SPLINE
SPL {X  -159.990, Y  +497.800, Z    +0.000, E1   +31.845, E3 +413374.245}
SPL {X  -159.990, Y  +492.180, Z    +0.000, E1   +32.851, E3 +413386.381}
SPL {X  -159.990, Y  +486.073, Z    +0.000, E1   +33.960, E3 +413399.016}
SPL {X  -159.990, Y  +477.314, Z    +0.000, E1   +35.342, E3 +413417.195}
SPL {X  -159.990, Y  +471.459, Z    +0.000, E1   +35.779, E3 +413431.734}
SPL {X  -159.990, Y  +467.485, Z    +0.000, E1   +35.768, E3 +413443.464}
SPL {X  -159.990, Y  +462.739, Z    +0.000, E1   +35.799, E3 +413457.392}
SPL {X  -159.990, Y  +457.385, Z    +0.000, E1   +35.788, E3 +413473.175}
SPL {X  -159.990, Y  +452.637, Z    +0.000, E1   +35.783, E3 +413487.167}
SPL {X  -159.990, Y  +448.227, Z    +0.000, E1   +35.776, E3 +413500.163}
SPL {X  -159.990, Y  +443.707, Z    +0.000, E1   +35.784, E3 +413513.459}
SPL {X  -159.990, Y  +439.109, Z    +0.000, E1   +35.781, E3 +413526.995}
SPL {X  -159.990, Y  +434.400, Z    +0.000, E1   +35.789, E3 +413540.849}
SPL {X  -159.990, Y  +430.115, Z    +0.000, E1   +35.777, E3 +413553.466}
SPL {X  -159.990, Y  +425.407, Z    +0.000, E1   +35.800, E3 +413567.306}
SPL {X  -159.990, Y  +420.199, Z    +0.000, E1   +35.790, E3 +413582.660}
SPL {X  -159.990, Y  +414.514, Z    +0.000, E1   +35.815, E3 +413599.359}
SPL {X  -159.990, Y  +408.600, Z    +0.000, E1   +35.802, E3 +413616.798}
SPL {X  -159.990, Y  +403.496, Z    +0.000, E1   +35.787, E3 +413631.852}
SPL {X  -159.990, Y  +398.606, Z    +0.000, E1   +35.794, E3 +413646.240}
SPL {X  -159.990, Y  +394.138, Z    +0.000, E1   +35.778, E3 +413659.423}
SPL {X  -159.990, Y  +388.813, Z    +0.000, E1   +35.819, E3 +413675.035}
SPL {X  -159.990, Y  +383.172, Z    +0.000, E1   +35.789, E3 +413691.689}
SPL {X  -159.936, Y  +378.352, Z    +0.000, E1   +35.782, E3 +413705.928}
SPL {X  -159.693, Y  +372.749, Z    +0.000, E1   +35.767, E3 +413722.660}
SPL {X  -159.203, Y  +366.647, Z    +0.000, E1   +35.680, E3 +413741.146}
SPL {X  -158.715, Y  +362.338, Z    +0.000, E1   +35.547, E3 +413754.451}
SPL {X  -158.237, Y  +358.884, Z    +0.000, E1   +35.480, E3 +413765.108}
SPL {X  -157.724, Y  +355.670, Z    +0.000, E1   +35.371, E3 +413775.142}
SPL {X  -157.185, Y  +352.671, Z    +0.000, E1   +35.292, E3 +413784.521}
SPL {X  -156.302, Y  +348.345, Z    +0.000, E1   +35.165, E3 +413798.142}
SPL {X  -155.054, Y  +343.066, Z    +0.000, E1   +34.964, E3 +413814.956}
SPL {X  -154.305, Y  +340.232, Z    +0.000, E1   +28.975, E3 +413872.516}
ENDSPLINE

SPLINE
SPL {X  -158.456, Y  +360.399, Z    +0.000, E1   +16.490, E3 +413909.336}
SPL {X  -159.553, Y  +370.677, Z    +0.000, E1   +10.576, E3 +413917.096}
SPL {X  -159.960, Y  +379.402, Z    +0.000, E1    +5.303, E3 +413921.116}
SPL {X  -159.990, Y  +387.301, Z    +0.000, E1    +0.001, E3 +413923.578}
SPL {X  -159.990, Y  +392.161, Z    +0.000, E1    -3.946, E3 +413924.989}
SPL {X  -159.990, Y  +396.375, Z    +0.000, E1    -7.538, E3 +413926.411}
SPL {X  -159.990, Y  +404.277, Z    +0.000, E1   -14.543, E3 +413930.075}
SPL {X  -159.990, Y  +423.101, Z    +0.000, E1   -27.351, E3 +413946.513}
SPL {X  -159.990, Y  +430.933, Z    +0.000, E1   -30.672, E3 +413956.484}
SPL {X  -159.990, Y  +451.842, Z    +0.000, E1   -35.050, E3 +413995.856}
SPL {X  -159.990, Y  +456.402, Z    +0.000, E1   -35.061, E3 +414009.632}
SPL {X  -159.990, Y  +460.708, Z    +0.000, E1   -35.045, E3 +414022.689}
SPL {X  -159.990, Y  +464.162, Z    +0.000, E1   -35.038, E3 +414033.146}
SPL {X  -159.990, Y  +467.857, Z    +0.000, E1   -35.053, E3 +414044.303}
SPL {X  -159.990, Y  +471.326, Z    +0.000, E1   -35.038, E3 +414054.798}
SPL {X  -159.990, Y  +474.610, Z    +0.000, E1   -35.053, E3 +414064.697}
SPL {X  -159.990, Y  +478.303, Z    +0.000, E1   -35.049, E3 +414075.869}
SPL {X  -159.990, Y  +482.537, Z    +0.000, E1   -35.066, E3 +414088.661}
SPL {X  -159.990, Y  +487.181, Z    +0.000, E1   -35.054, E3 +414102.744}
SPL {X  -159.990, Y  +492.368, Z    +0.000, E1   -35.076, E3 +414118.415}
SPL {X  -159.990, Y  +497.072, Z    +0.000, E1   -35.040, E3 +414132.712}
SPL {X  -159.990, Y  +501.645, Z    +0.000, E1   -35.067, E3 +414146.495}
SPL {X  -159.990, Y  +506.307, Z    +0.000, E1   -35.049, E3 +414160.617}
SPL {X  -159.990, Y  +511.643, Z    +0.000, E1   -35.091, E3 +414176.697}
SPL {X  -159.990, Y  +517.156, Z    +0.000, E1   -35.059, E3 +414193.415}
SPL {X  -159.990, Y  +521.637, Z    +0.000, E1   -35.056, E3 +414206.978}
SPL {X  -159.990, Y  +526.246, Z    +0.000, E1   -35.065, E3 +414220.882}
SPL {X  -159.990, Y  +530.289, Z    +0.000, E1   -35.044, E3 +414233.168}
SPL {X  -159.990, Y  +534.797, Z    +0.000, E1   -35.069, E3 +414246.768}
SPL {X  -159.990, Y  +538.710, Z    +0.000, E1   -35.033, E3 +414258.665}
SPL {X  -159.990, Y  +542.114, Z    +0.000, E1   -35.053, E3 +414268.917}
SPL {X  -159.990, Y  +545.724, Z    +0.000, E1   -35.043, E3 +414279.842}
SPL {X  -159.990, Y  +549.546, Z    +0.000, E1   -35.061, E3 +414291.366}
SPL {X  -159.990, Y  +554.793, Z    +0.000, E1   -35.100, E3 +414307.129}
SPL {X  -159.990, Y  +560.931, Z    +0.000, E1   -35.098, E3 +414325.691}
SPL {X  -159.990, Y  +566.542, Z    +0.000, E1   -35.080, E3 +414342.699}
SPL {X  -159.990, Y  +570.261, Z    +0.000, E1   -35.046, E3 +414353.995}
SPL {X  -159.990, Y  +574.780, Z    +0.000, E1   -35.101, E3 +414367.574}
SPL {X  -159.990, Y  +580.750, Z    +0.000, E1   -35.087, E3 +414385.650}
SPL {X  -159.990, Y  +585.414, Z    +0.000, E1   -35.059, E3 +414399.796}
SPL {X  -159.990, Y  +588.716, Z    +0.000, E1   -35.047, E3 +414409.799}
SPL {X  -159.990, Y  +592.923, Z    +0.000, E1   -35.084, E3 +414422.463}
SPL {X  -159.990, Y  +598.554, Z    +0.000, E1   -35.088, E3 +414439.483}
SPL {X  -159.990, Y  +603.289, Z    +0.000, E1   -35.068, E3 +414453.810}
SPL {X  -159.990, Y  +606.793, Z    +0.000, E1   -35.050, E3 +414464.452}
SPL {X  -159.990, Y  +611.113, Z    +0.000, E1   -35.087, E3 +414477.443}
SPL {X  -159.990, Y  +616.690, Z    +0.000, E1   -35.089, E3 +414494.306}
SPL {X  -159.990, Y  +621.534, Z    +0.000, E1   -35.068, E3 +414508.965}
SPL {X  -159.990, Y  +625.237, Z    +0.000, E1   -35.062, E3 +414520.167}
SPL {X  -159.990, Y  +629.217, Z    +0.000, E1   -35.065, E3 +414532.225}
SPL {X  -159.990, Y  +632.566, Z    +0.000, E1   -35.044, E3 +414542.387}
SPL {X  -159.990, Y  +636.917, Z    +0.000, E1   -35.095, E3 +414555.462}
SPL {X  -159.990, Y  +641.534, Z    +0.000, E1   -35.053, E3 +414569.489}
SPL {X  -159.990, Y  +645.423, Z    +0.000, E1   -35.070, E3 +414581.225}
SPL {X  -159.990, Y  +650.555, Z    +0.000, E1   -35.089, E3 +414596.714}
SPL {X  -159.990, Y  +656.270, Z    +0.000, E1   -35.087, E3 +414614.007}
SPL {X  -159.990, Y  +661.105, Z    +0.000, E1   -35.059, E3 +414628.671}
SPL {X  -159.990, Y  +665.311, Z    +0.000, E1   -35.064, E3 +414641.385}
SPL {X  -159.990, Y  +670.193, Z    +0.000, E1   -35.076, E3 +414656.133}
SPL {X  -159.948, Y  +675.148, Z    +0.000, E1   -35.069, E3 +414671.125}
SPL {X  -159.805, Y  +679.202, Z    +0.000, E1   -35.029, E3 +414683.557}
SPL {X  -159.584, Y  +682.885, Z    +0.000, E1   -34.997, E3 +414694.917}
SPL {X  -159.292, Y  +686.426, Z    +0.000, E1   -34.947, E3 +414705.919}
SPL {X  -158.886, Y  +690.264, Z    +0.000, E1   -34.888, E3 +414717.935}
SPL {X  -158.362, Y  +694.266, Z    +0.000, E1   -34.794, E3 +414730.609}
SPL {X  -157.614, Y  +698.973, Z    +0.000, E1   -34.690, E3 +414745.609}
SPL {X  -156.640, Y  +704.066, Z    +0.000, E1   -34.516, E3 +414762.034}
SPL {X  -155.835, Y  +707.723, Z    +0.000, E1   -34.344, E3 +414773.977}
SPL {X  -155.153, Y  +710.542, Z    +0.000, E1   -34.234, E3 +414783.196}
SPL {X  -153.767, Y  +715.686, Z    +0.000, E1   -30.747, E3 +414828.414}
ENDSPLINE

SPLINE
SPL {X  -155.537, Y  +708.983, Z    +0.000, E1   -25.008, E3 +414859.219}
SPL {X  -158.838, Y  +690.666, Z    +0.000, E1   -14.584, E3 +414883.932}
SPL {X  -159.750, Y  +680.262, Z    +0.000, E1    -8.563, E3 +414890.072}
SPL {X  -159.973, Y  +673.798, Z    +0.000, E1    -4.600, E3 +414892.536}
SPL {X  -159.990, Y  +667.448, Z    +0.000, E1    -0.356, E3 +414894.316}
SPL {X  -159.990, Y  +662.686, Z    +0.000, E1    +3.472, E3 +414895.551}
SPL {X  -159.990, Y  +657.071, Z    +0.000, E1    +8.297, E3 +414897.429}
SPL {X  -159.990, Y  +646.193, Z    +0.000, E1   +17.980, E3 +414903.156}
SPL {X  -159.990, Y  +621.124, Z    +0.000, E1   +32.598, E3 +414926.643}
SPL {X  -159.990, Y  +597.855, Z    +0.000, E1   +36.862, E3 +414969.562}
SPL {X  -159.990, Y  +592.884, Z    +0.000, E1   +36.865, E3 +414983.633}
SPL {X  -159.990, Y  +587.104, Z    +0.000, E1   +36.878, E3 +414999.990}
SPL {X  -159.990, Y  +581.795, Z    +0.000, E1   +36.847, E3 +415015.088}
SPL {X  -159.990, Y  +577.286, Z    +0.000, E1   +36.853, E3 +415027.845}
SPL {X  -159.990, Y  +572.409, Z    +0.000, E1   +36.854, E3 +415041.657}
SPL {X  -159.990, Y  +567.110, Z    +0.000, E1   +36.868, E3 +415056.619}
SPL {X  -159.990, Y  +562.387, Z    +0.000, E1   +36.853, E3 +415069.980}
SPL {X  -159.990, Y  +557.944, Z    +0.000, E1   +36.859, E3 +415082.574}
SPL {X  -159.990, Y  +553.661, Z    +0.000, E1   +36.844, E3 +415094.737}
SPL {X  -159.990, Y  +549.195, Z    +0.000, E1   +36.856, E3 +415107.373}
SPL {X  -159.990, Y  +544.733, Z    +0.000, E1   +36.845, E3 +415120.019}
SPL {X  -159.990, Y  +539.889, Z    +0.000, E1   +36.872, E3 +415133.703}
SPL {X  -159.990, Y  +534.469, Z    +0.000, E1   +36.855, E3 +415149.101}
SPL {X  -159.990, Y  +530.428, Z    +0.000, E1   +36.821, E3 +415160.634}
SPL {X  -159.990, Y  +527.151, Z    +0.000, E1   +36.828, E3 +415169.897}
SPL {X  -159.990, Y  +522.641, Z    +0.000, E1   +36.854, E3 +415182.629}
SPL {X  -159.990, Y  +517.225, Z    +0.000, E1   +36.859, E3 +415197.964}
SPL {X  -159.990, Y  +512.789, Z    +0.000, E1   +36.824, E3 +415210.591}
SPL {X  -159.990, Y  +508.591, Z    +0.000, E1   +36.846, E3 +415222.454}
SPL {X  -159.990, Y  +503.454, Z    +0.000, E1   +36.847, E3 +415237.009}
SPL {X  -159.990, Y  +498.507, Z    +0.000, E1   +36.487, E3 +415253.458}
ENDSPLINE

SPLINE
SPL {X  -159.990, Y  +506.994, Z    +0.000, E1   +30.162, E3 +415265.967}
ENDSPLINE

SPLINE
SPL {X  -159.990, Y  +502.084, Z    +0.000, E1   +31.057, E3 +415277.619}
SPL {X  -159.990, Y  +496.272, Z    +0.000, E1   +32.117, E3 +415290.610}
SPL {X  -159.990, Y  +492.180, Z    +0.000, E1   +32.851, E3 +415299.424}
SPL {X  -159.990, Y  +486.073, Z    +0.000, E1   +33.960, E3 +415312.060}
SPL {X  -159.990, Y  +477.314, Z    +0.000, E1   +35.342, E3 +415330.238}
SPL {X  -159.990, Y  +471.459, Z    +0.000, E1   +35.779, E3 +415344.778}
SPL {X  -159.990, Y  +467.485, Z    +0.000, E1   +35.768, E3 +415356.507}
SPL {X  -159.990, Y  +462.739, Z    +0.000, E1   +35.799, E3 +415370.435}
SPL {X  -159.990, Y  +457.385, Z    +0.000, E1   +35.788, E3 +415386.218}
SPL {X  -159.990, Y  +452.637, Z    +0.000, E1   +35.783, E3 +415400.210}
SPL {X  -159.990, Y  +448.227, Z    +0.000, E1   +35.776, E3 +415413.207}
SPL {X  -159.990, Y  +443.707, Z    +0.000, E1   +35.784, E3 +415426.502}
SPL {X  -159.990, Y  +439.109, Z    +0.000, E1   +35.781, E3 +415440.038}
SPL {X  -159.990, Y  +435.535, Z    +0.000, E1   +35.764, E3 +415450.589}
SPL {X  -159.990, Y  +431.100, Z    +0.000, E1   +35.807, E3 +415463.574}
SPL {X  -159.990, Y  +426.641, Z    +0.000, E1   +35.769, E3 +415476.760}
SPL {X  -159.990, Y  +422.627, Z    +0.000, E1   +35.788, E3 +415488.558}
SPL {X  -159.990, Y  +419.027, Z    +0.000, E1   +35.762, E3 +415499.198}
SPL {X  -159.990, Y  +414.514, Z    +0.000, E1   +35.815, E3 +415512.402}
SPL {X  -159.990, Y  +409.702, Z    +0.000, E1   +35.772, E3 +415526.643}
SPL {X  -159.990, Y  +404.413, Z    +0.000, E1   +35.821, E3 +415542.146}
SPL {X  -159.990, Y  +398.606, Z    +0.000, E1   +35.794, E3 +415559.283}
SPL {X  -159.990, Y  +394.138, Z    +0.000, E1   +35.778, E3 +415572.466}
SPL {X  -159.990, Y  +388.813, Z    +0.000, E1   +35.819, E3 +415588.078}
SPL {X  -159.990, Y  +383.172, Z    +0.000, E1   +35.789, E3 +415604.733}
SPL {X  -159.936, Y  +378.352, Z    +0.000, E1   +35.782, E3 +415618.972}
SPL {X  -159.790, Y  +374.497, Z    +0.000, E1   +35.735, E3 +415630.516}
SPL {X  -159.547, Y  +370.604, Z    +0.000, E1   +35.724, E3 +415642.201}
SPL {X  -159.134, Y  +365.969, Z    +0.000, E1   +35.644, E3 +415656.286}
SPL {X  -158.606, Y  +361.498, Z    +0.000, E1   +35.550, E3 +415670.051}
SPL {X  -157.918, Y  +356.833, Z    +0.000, E1   +35.439, E3 +415684.503}
SPL {X  -157.185, Y  +352.671, Z    +0.000, E1   +35.292, E3 +415697.564}
SPL {X  -156.302, Y  +348.345, Z    +0.000, E1   +35.165, E3 +415711.185}
SPL {X  -155.054, Y  +343.066, Z    +0.000, E1   +34.964, E3 +415728.000}
SPL {X  -154.305, Y  +340.232, Z    +0.000, E1   +28.975, E3 +415785.560}
ENDSPLINE

SPLINE
SPL {X  -158.456, Y  +360.399, Z    +0.000, E1   +16.490, E3 +415822.380}
SPL {X  -159.553, Y  +370.677, Z    +0.000, E1   +10.576, E3 +415830.140}
SPL {X  -159.960, Y  +379.402, Z    +0.000, E1    +5.303, E3 +415834.160}
SPL {X  -159.990, Y  +387.301, Z    +0.000, E1    +0.001, E3 +415836.621}
SPL {X  -159.990, Y  +392.161, Z    +0.000, E1    -3.946, E3 +415838.033}
SPL {X  -159.990, Y  +396.375, Z    +0.000, E1    -7.538, E3 +415839.455}
SPL {X  -159.990, Y  +404.277, Z    +0.000, E1   -14.543, E3 +415843.118}
SPL {X  -159.990, Y  +423.101, Z    +0.000, E1   -27.351, E3 +415859.557}
SPL {X  -159.990, Y  +430.933, Z    +0.000, E1   -30.672, E3 +415869.528}
SPL {X  -159.990, Y  +451.842, Z    +0.000, E1   -35.050, E3 +415908.899}
SPL {X  -159.990, Y  +456.402, Z    +0.000, E1   -35.061, E3 +415922.675}
SPL {X  -159.990, Y  +460.708, Z    +0.000, E1   -35.045, E3 +415935.733}
SPL {X  -159.990, Y  +464.162, Z    +0.000, E1   -35.038, E3 +415946.189}
SPL {X  -159.990, Y  +467.857, Z    +0.000, E1   -35.053, E3 +415957.346}
SPL {X  -159.990, Y  +471.326, Z    +0.000, E1   -35.038, E3 +415967.841}
SPL {X  -159.990, Y  +474.610, Z    +0.000, E1   -35.053, E3 +415977.741}
SPL {X  -159.990, Y  +478.303, Z    +0.000, E1   -35.049, E3 +415988.913}
SPL {X  -159.990, Y  +482.537, Z    +0.000, E1   -35.066, E3 +416001.704}
SPL {X  -159.990, Y  +487.181, Z    +0.000, E1   -35.054, E3 +416015.787}
SPL {X  -159.990, Y  +490.807, Z    +0.000, E1   -35.036, E3 +416026.788}
SPL {X  -159.990, Y  +493.669, Z    +0.000, E1   -35.034, E3 +416035.468}
SPL {X  -159.990, Y  +497.072, Z    +0.000, E1   -35.040, E3 +416045.755}
SPL {X  -159.990, Y  +501.645, Z    +0.000, E1   -35.067, E3 +416059.538}
SPL {X  -159.990, Y  +507.359, Z    +0.000, E1   -35.080, E3 +416076.795}
SPL {X  -159.990, Y  +512.562, Z    +0.000, E1   -35.055, E3 +416092.577}
SPL {X  -159.990, Y  +517.156, Z    +0.000, E1   -35.059, E3 +416106.458}
SPL {X  -159.990, Y  +521.637, Z    +0.000, E1   -35.056, E3 +416120.022}
SPL {X  -159.990, Y  +525.227, Z    +0.000, E1   -35.041, E3 +416130.882}
SPL {X  -159.990, Y  +529.413, Z    +0.000, E1   -35.072, E3 +416143.511}
SPL {X  -159.990, Y  +534.797, Z    +0.000, E1   -35.069, E3 +416159.812}
SPL {X  -159.990, Y  +538.710, Z    +0.000, E1   -35.033, E3 +416171.709}
SPL {X  -159.990, Y  +542.114, Z    +0.000, E1   -35.053, E3 +416181.961}
SPL {X  -159.990, Y  +546.612, Z    +0.000, E1   -35.065, E3 +416195.532}
SPL {X  -159.990, Y  +551.596, Z    +0.000, E1   -35.079, E3 +416210.567}
SPL {X  -159.990, Y  +557.043, Z    +0.000, E1   -35.087, E3 +416226.989}
SPL {X  -159.990, Y  +562.842, Z    +0.000, E1   -35.098, E3 +416244.522}
SPL {X  -159.990, Y  +568.750, Z    +0.000, E1   -35.087, E3 +416262.407}
SPL {X  -159.990, Y  +574.780, Z    +0.000, E1   -35.101, E3 +416280.618}
SPL {X  -159.990, Y  +580.750, Z    +0.000, E1   -35.087, E3 +416298.694}
SPL {X  -159.990, Y  +585.414, Z    +0.000, E1   -35.059, E3 +416312.840}
SPL {X  -159.990, Y  +588.716, Z    +0.000, E1   -35.047, E3 +416322.843}
SPL {X  -159.990, Y  +592.923, Z    +0.000, E1   -35.084, E3 +416335.507}
SPL {X  -159.990, Y  +598.554, Z    +0.000, E1   -35.088, E3 +416352.526}
SPL {X  -159.990, Y  +603.289, Z    +0.000, E1   -35.068, E3 +416366.854}
SPL {X  -159.990, Y  +607.919, Z    +0.000, E1   -35.079, E3 +416380.842}
SPL {X  -159.990, Y  +613.036, Z    +0.000, E1   -35.082, E3 +416396.313}
SPL {X  -159.990, Y  +617.577, Z    +0.000, E1   -35.061, E3 +416410.075}
SPL {X  -159.990, Y  +621.534, Z    +0.000, E1   -35.068, E3 +416422.009}
SPL {X  -159.990, Y  +626.426, Z    +0.000, E1   -35.093, E3 +416436.768}
SPL {X  -159.990, Y  +631.553, Z    +0.000, E1   -35.068, E3 +416452.326}
SPL {X  -159.990, Y  +636.917, Z    +0.000, E1   -35.095, E3 +416468.505}
SPL {X  -159.990, Y  +641.534, Z    +0.000, E1   -35.053, E3 +416482.533}
SPL {X  -159.990, Y  +646.430, Z    +0.000, E1   -35.102, E3 +416497.264}
SPL {X  -159.990, Y  +651.502, Z    +0.000, E1   -35.058, E3 +416512.674}
SPL {X  -159.990, Y  +654.793, Z    +0.000, E1   -35.049, E3 +416522.637}
SPL {X  -159.990, Y  +657.535, Z    +0.000, E1   -35.049, E3 +416530.934}
SPL {X  -159.990, Y  +661.105, Z    +0.000, E1   -35.059, E3 +416541.714}
SPL {X  -159.990, Y  +665.311, Z    +0.000, E1   -35.064, E3 +416554.429}
SPL {X  -159.990, Y  +670.193, Z    +0.000, E1   -35.076, E3 +416569.176}
SPL {X  -159.948, Y  +675.148, Z    +0.000, E1   -35.069, E3 +416584.168}
SPL {X  -159.752, Y  +680.228, Z    +0.000, E1   -35.050, E3 +416599.716}
SPL {X  -159.371, Y  +685.563, Z    +0.000, E1   -34.989, E3 +416616.227}
SPL {X  -158.886, Y  +690.264, Z    +0.000, E1   -34.888, E3 +416630.979}
SPL {X  -158.362, Y  +694.266, Z    +0.000, E1   -34.794, E3 +416643.652}
SPL {X  -157.614, Y  +698.973, Z    +0.000, E1   -34.690, E3 +416658.653}
SPL {X  -156.640, Y  +704.066, Z    +0.000, E1   -34.516, E3 +416675.078}
SPL {X  -155.835, Y  +707.723, Z    +0.000, E1   -34.344, E3 +416687.020}
SPL {X  -155.080, Y  +710.833, Z    +0.000, E1   -34.231, E3 +416697.170}
SPL {X  -153.755, Y  +715.731, Z    +0.000, E1   -30.246, E3 +416746.436}
ENDSPLINE

SPLINE
SPL {X  -155.537, Y  +708.983, Z    +0.000, E1   -25.008, E3 +416772.263}
SPL {X  -158.838, Y  +690.666, Z    +0.000, E1   -14.584, E3 +416796.975}
SPL {X  -159.750, Y  +680.262, Z    +0.000, E1    -8.563, E3 +416803.116}
SPL {X  -159.973, Y  +673.798, Z    +0.000, E1    -4.600, E3 +416805.580}
SPL {X  -159.990, Y  +668.863, Z    +0.000, E1    -1.298, E3 +416807.019}
SPL {X  -159.990, Y  +663.839, Z    +0.000, E1    +2.454, E3 +416808.280}
SPL {X  -159.990, Y  +657.071, Z    +0.000, E1    +8.297, E3 +416810.473}
SPL {X  -159.990, Y  +646.193, Z    +0.000, E1   +17.980, E3 +416816.199}
SPL {X  -159.990, Y  +621.124, Z    +0.000, E1   +32.598, E3 +416839.686}
SPL {X  -159.990, Y  +597.855, Z    +0.000, E1   +36.862, E3 +416882.605}
SPL {X  -159.990, Y  +592.884, Z    +0.000, E1   +36.865, E3 +416896.676}
SPL {X  -159.990, Y  +587.104, Z    +0.000, E1   +36.878, E3 +416913.033}
SPL {X  -159.990, Y  +581.795, Z    +0.000, E1   +36.847, E3 +416928.132}
SPL {X  -159.990, Y  +577.286, Z    +0.000, E1   +36.853, E3 +416940.889}
SPL {X  -159.990, Y  +572.409, Z    +0.000, E1   +36.854, E3 +416954.701}
SPL {X  -159.990, Y  +567.110, Z    +0.000, E1   +36.868, E3 +416969.662}
SPL {X  -159.990, Y  +562.387, Z    +0.000, E1   +36.853, E3 +416983.023}
SPL {X  -159.990, Y  +557.944, Z    +0.000, E1   +36.859, E3 +416995.617}
SPL {X  -159.990, Y  +553.661, Z    +0.000, E1   +36.844, E3 +417007.781}
SPL {X  -159.990, Y  +549.195, Z    +0.000, E1   +36.856, E3 +417020.416}
SPL {X  -159.990, Y  +544.733, Z    +0.000, E1   +36.845, E3 +417033.062}
SPL {X  -159.990, Y  +539.889, Z    +0.000, E1   +36.872, E3 +417046.746}
SPL {X  -159.990, Y  +534.469, Z    +0.000, E1   +36.855, E3 +417062.144}
SPL {X  -159.990, Y  +530.428, Z    +0.000, E1   +36.821, E3 +417073.678}
SPL {X  -159.990, Y  +525.940, Z    +0.000, E1   +36.859, E3 +417086.324}
SPL {X  -159.990, Y  +520.301, Z    +0.000, E1   +36.855, E3 +417102.300}
SPL {X  -159.990, Y  +514.308, Z    +0.000, E1   +36.869, E3 +417119.262}
SPL {X  -159.990, Y  +508.591, Z    +0.000, E1   +36.846, E3 +417135.497}
SPL {X  -159.990, Y  +503.454, Z    +0.000, E1   +36.847, E3 +417150.052}
SPL {X  -159.990, Y  +498.507, Z    +0.000, E1   +36.487, E3 +417166.501}
ENDSPLINE

SPLINE
SPL {X  -159.990, Y  +506.994, Z    +0.000, E1   +30.162, E3 +417179.011}
ENDSPLINE

SPLINE
SPL {X  -159.990, Y  +502.084, Z    +0.000, E1   +31.057, E3 +417190.662}
SPL {X  -159.990, Y  +494.586, Z    +0.000, E1   +32.444, E3 +417207.265}
SPL {X  -159.990, Y  +487.723, Z    +0.000, E1   +33.658, E3 +417221.718}
SPL {X  -159.990, Y  +481.374, Z    +0.000, E1   +34.706, E3 +417234.922}
SPL {X  -159.990, Y  +475.503, Z    +0.000, E1   +35.597, E3 +417246.975}
SPL {X  -159.990, Y  +471.459, Z    +0.000, E1   +35.779, E3 +417257.821}
SPL {X  -159.990, Y  +467.485, Z    +0.000, E1   +35.768, E3 +417269.551}
SPL {X  -159.990, Y  +462.739, Z    +0.000, E1   +35.799, E3 +417283.478}
SPL {X  -159.990, Y  +457.385, Z    +0.000, E1   +35.788, E3 +417299.262}
SPL {X  -159.990, Y  +452.637, Z    +0.000, E1   +35.783, E3 +417313.254}
SPL {X  -159.990, Y  +448.227, Z    +0.000, E1   +35.776, E3 +417326.250}
SPL {X  -159.990, Y  +443.707, Z    +0.000, E1   +35.784, E3 +417339.546}
SPL {X  -159.990, Y  +439.109, Z    +0.000, E1   +35.781, E3 +417353.082}
SPL {X  -159.990, Y  +434.400, Z    +0.000, E1   +35.789, E3 +417366.936}
SPL {X  -159.990, Y  +430.115, Z    +0.000, E1   +35.777, E3 +417379.553}
SPL {X  -159.990, Y  +425.407, Z    +0.000, E1   +35.800, E3 +417393.393}
SPL {X  -159.990, Y  +420.199, Z    +0.000, E1   +35.790, E3 +417408.747}
SPL {X  -159.990, Y  +414.514, Z    +0.000, E1   +35.815, E3 +417425.446}
SPL {X  -159.990, Y  +409.702, Z    +0.000, E1   +35.772, E3 +417439.687}
SPL {X  -159.990, Y  +405.848, Z    +0.000, E1   +35.776, E3 +417451.033}
SPL {X  -159.990, Y  +400.924, Z    +0.000, E1   +35.804, E3 +417465.491}
SPL {X  -159.990, Y  +395.017, Z    +0.000, E1   +35.806, E3 +417482.879}
SPL {X  -159.990, Y  +390.065, Z    +0.000, E1   +35.780, E3 +417497.500}
SPL {X  -159.990, Y  +385.506, Z    +0.000, E1   +35.789, E3 +417510.906}
SPL {X  -159.976, Y  +380.359, Z    +0.000, E1   +35.797, E3 +417526.055}
SPL {X  -159.831, Y  +375.358, Z    +0.000, E1   +35.763, E3 +417540.945}
SPL {X  -159.547, Y  +370.604, Z    +0.000, E1   +35.724, E3 +417555.244}
SPL {X  -159.134, Y  +365.969, Z    +0.000, E1   +35.644, E3 +417569.330}
SPL {X  -158.715, Y  +362.338, Z    +0.000, E1   +35.547, E3 +417580.538}
SPL {X  -158.237, Y  +358.884, Z    +0.000, E1   +35.480, E3 +417591.195}
SPL {X  -157.724, Y  +355.670, Z    +0.000, E1   +35.371, E3 +417601.229}
SPL {X  -157.185, Y  +352.671, Z    +0.000, E1   +35.292, E3 +417610.608}
SPL {X  -156.582, Y  +349.653, Z    +0.000, E1   +35.175, E3 +417620.141}
SPL {X  -155.743, Y  +345.880, Z    +0.000, E1   +35.068, E3 +417632.068}
SPL {X  -154.759, Y  +341.925, Z    +0.000, E1   +34.868, E3 +417644.774}
SPL {X  -154.305, Y  +340.232, Z    +0.000, E1   +28.975, E3 +417698.603}
ENDSPLINE

SPLINE
SPL {X  -158.456, Y  +360.399, Z    +0.000, E1   +16.490, E3 +417735.423}
SPL {X  -159.553, Y  +370.677, Z    +0.000, E1   +10.576, E3 +417743.183}
SPL {X  -159.960, Y  +379.402, Z    +0.000, E1    +5.303, E3 +417747.203}
SPL {X  -159.990, Y  +385.983, Z    +0.000, E1    +0.882, E3 +417749.276}
SPL {X  -159.990, Y  +390.933, Z    +0.000, E1    -2.877, E3 +417750.724}
SPL {X  -159.990, Y  +396.375, Z    +0.000, E1    -7.538, E3 +417752.498}
SPL {X  -159.990, Y  +404.277, Z    +0.000, E1   -14.543, E3 +417756.162}
SPL {X  -159.990, Y  +423.101, Z    +0.000, E1   -27.351, E3 +417772.600}
SPL {X  -159.990, Y  +430.933, Z    +0.000, E1   -30.672, E3 +417782.571}
SPL {X  -159.990, Y  +452.779, Z    +0.000, E1   -35.077, E3 +417824.734}
SPL {X  -159.990, Y  +457.209, Z    +0.000, E1   -35.039, E3 +417838.194}
SPL {X  -159.990, Y  +460.708, Z    +0.000, E1   -35.045, E3 +417848.776}
SPL {X  -159.990, Y  +465.240, Z    +0.000, E1   -35.066, E3 +417862.452}
SPL {X  -159.990, Y  +470.278, Z    +0.000, E1   -35.063, E3 +417877.685}
SPL {X  -159.990, Y  +474.610, Z    +0.000, E1   -35.053, E3 +417890.784}
SPL {X  -159.990, Y  +478.303, Z    +0.000, E1   -35.049, E3 +417901.956}
SPL {X  -159.990, Y  +482.537, Z    +0.000, E1   -35.066, E3 +417914.748}
SPL {X  -159.990, Y  +487.181, Z    +0.000, E1   -35.054, E3 +417928.830}
SPL {X  -159.990, Y  +492.368, Z    +0.000, E1   -35.076, E3 +417944.502}
SPL {X  -159.990, Y  +497.072, Z    +0.000, E1   -35.040, E3 +417958.799}
SPL {X  -159.990, Y  +501.645, Z    +0.000, E1   -35.067, E3 +417972.582}
SPL {X  -159.990, Y  +507.359, Z    +0.000, E1   -35.080, E3 +417989.838}
SPL {X  -159.990, Y  +512.562, Z    +0.000, E1   -35.055, E3 +418005.620}
SPL {X  -159.990, Y  +517.156, Z    +0.000, E1   -35.059, E3 +418019.502}
SPL {X  -159.990, Y  +521.637, Z    +0.000, E1   -35.056, E3 +418033.065}
SPL {X  -159.990, Y  +526.246, Z    +0.000, E1   -35.065, E3 +418046.969}
SPL {X  -159.990, Y  +531.319, Z    +0.000, E1   -35.072, E3 +418062.325}
SPL {X  -159.990, Y  +537.053, Z    +0.000, E1   -35.083, E3 +418079.657}
SPL {X  -159.990, Y  +542.114, Z    +0.000, E1   -35.053, E3 +418095.004}
SPL {X  -159.990, Y  +546.612, Z    +0.000, E1   -35.065, E3 +418108.576}
SPL {X  -159.990, Y  +551.596, Z    +0.000, E1   -35.079, E3 +418123.611}
SPL {X  -159.990, Y  +557.043, Z    +0.000, E1   -35.087, E3 +418140.032}
SPL {X  -159.990, Y  +561.808, Z    +0.000, E1   -35.066, E3 +418154.486}
SPL {X  -159.990, Y  +566.542, Z    +0.000, E1   -35.080, E3 +418168.786}
SPL {X  -159.990, Y  +571.374, Z    +0.000, E1   -35.070, E3 +418183.409}
SPL {X  -159.990, Y  +575.771, Z    +0.000, E1   -35.064, E3 +418196.715}
SPL {X  -159.990, Y  +580.750, Z    +0.000, E1   -35.087, E3 +418211.737}
SPL {X  -159.990, Y  +585.414, Z    +0.000, E1   -35.059, E3 +418225.883}
SPL {X  -159.990, Y  +590.166, Z    +0.000, E1   -35.084, E3 +418240.212}
SPL {X  -159.990, Y  +595.313, Z    +0.000, E1   -35.073, E3 +418255.790}
SPL {X  -159.990, Y  +600.543, Z    +0.000, E1   -35.091, E3 +418271.573}
SPL {X  -159.990, Y  +605.846, Z    +0.000, E1   -35.077, E3 +418287.624}
SPL {X  -159.990, Y  +611.113, Z    +0.000, E1   -35.087, E3 +418303.530}
SPL {X  -159.990, Y  +616.690, Z    +0.000, E1   -35.089, E3 +418320.393}
SPL {X  -159.990, Y  +621.534, Z    +0.000, E1   -35.068, E3 +418335.052}
SPL {X  -159.990, Y  +626.426, Z    +0.000, E1   -35.093, E3 +418349.812}
SPL {X  -159.990, Y  +631.553, Z    +0.000, E1   -35.068, E3 +418365.370}
SPL {X  -159.990, Y  +635.965, Z    +0.000, E1   -35.065, E3 +418378.718}
SPL {X  -159.990, Y  +640.633, Z    +0.000, E1   -35.080, E3 +418392.806}
SPL {X  -159.990, Y  +645.423, Z    +0.000, E1   -35.070, E3 +418407.312}
SPL {X  -159.990, Y  +650.555, Z    +0.000, E1   -35.089, E3 +418422.801}
SPL {X  -159.990, Y  +656.270, Z    +0.000, E1   -35.087, E3 +418440.094}
SPL {X  -159.990, Y  +661.105, Z    +0.000, E1   -35.059, E3 +418454.758}
SPL {X  -159.990, Y  +665.311, Z    +0.000, E1   -35.064, E3 +418467.472}
SPL {X  -159.990, Y  +670.193, Z    +0.000, E1   -35.076, E3 +418482.220}
SPL {X  -159.948, Y  +675.148, Z    +0.000, E1   -35.069, E3 +418497.212}
SPL {X  -159.752, Y  +680.228, Z    +0.000, E1   -35.050, E3 +418512.759}
SPL {X  -159.371, Y  +685.563, Z    +0.000, E1   -34.989, E3 +418529.271}
SPL {X  -158.886, Y  +690.264, Z    +0.000, E1   -34.888, E3 +418544.022}
SPL {X  -158.362, Y  +694.266, Z    +0.000, E1   -34.794, E3 +418556.696}
SPL {X  -157.880, Y  +697.401, Z    +0.000, E1   -34.689, E3 +418566.730}
SPL {X  -157.427, Y  +700.022, Z    +0.000, E1   -34.620, E3 +418575.120}
SPL {X  -156.640, Y  +704.066, Z    +0.000, E1   -34.516, E3 +418588.121}
SPL {X  -155.835, Y  +707.723, Z    +0.000, E1   -34.344, E3 +418600.064}
SPL {X  -155.080, Y  +710.833, Z    +0.000, E1   -34.231, E3 +418610.214}
SPL {X  -153.755, Y  +715.731, Z    +0.000, E1   -30.246, E3 +418659.480}
ENDSPLINE

SPLINE
SPL {X  -155.537, Y  +708.983, Z    +0.000, E1   -25.008, E3 +418685.306}
SPL {X  -158.838, Y  +690.666, Z    +0.000, E1   -14.584, E3 +418710.019}
SPL {X  -159.750, Y  +680.262, Z    +0.000, E1    -8.563, E3 +418716.159}
SPL {X  -159.973, Y  +673.798, Z    +0.000, E1    -4.600, E3 +418718.623}
SPL {X  -159.990, Y  +667.448, Z    +0.000, E1    -0.356, E3 +418720.403}
SPL {X  -159.990, Y  +662.686, Z    +0.000, E1    +3.472, E3 +418721.638}
SPL {X  -159.990, Y  +657.071, Z    +0.000, E1    +8.297, E3 +418723.516}
SPL {X  -159.990, Y  +646.193, Z    +0.000, E1   +17.980, E3 +418729.243}
SPL {X  -159.990, Y  +621.124, Z    +0.000, E1   +32.598, E3 +418752.729}
SPL {X  -159.990, Y  +597.855, Z    +0.000, E1   +36.862, E3 +418795.649}
SPL {X  -159.990, Y  +592.884, Z    +0.000, E1   +36.865, E3 +418809.720}
SPL {X  -159.990, Y  +587.104, Z    +0.000, E1   +36.878, E3 +418826.076}
SPL {X  -159.990, Y  +581.795, Z    +0.000, E1   +36.847, E3 +418841.175}
SPL {X  -159.990, Y  +576.165, Z    +0.000, E1   +36.887, E3 +418857.055}
SPL {X  -159.990, Y  +570.328, Z    +0.000, E1   +36.855, E3 +418873.628}
SPL {X  -159.990, Y  +566.126, Z    +0.000, E1   +36.841, E3 +418885.534}
SPL {X  -159.990, Y  +562.387, Z    +0.000, E1   +36.853, E3 +418896.067}
SPL {X  -159.990, Y  +557.944, Z    +0.000, E1   +36.859, E3 +418908.661}
SPL {X  -159.990, Y  +553.661, Z    +0.000, E1   +36.844, E3 +418920.824}
SPL {X  -159.990, Y  +549.195, Z    +0.000, E1   +36.856, E3 +418933.460}
SPL {X  -159.990, Y  +543.458, Z    +0.000, E1   +36.882, E3 +418949.658}
SPL {X  -159.990, Y  +537.639, Z    +0.000, E1   +36.860, E3 +418966.196}
SPL {X  -159.990, Y  +531.894, Z    +0.000, E1   +36.865, E3 +418982.485}
SPL {X  -159.990, Y  +525.940, Z    +0.000, E1   +36.859, E3 +418999.367}
SPL {X  -159.990, Y  +520.301, Z    +0.000, E1   +36.855, E3 +419015.344}
SPL {X  -159.990, Y  +516.005, Z    +0.000, E1   +36.824, E3 +419027.570}
SPL {X  -159.990, Y  +511.408, Z    +0.000, E1   +36.858, E3 +419040.539}
SPL {X  -159.990, Y  +505.756, Z    +0.000, E1   +36.857, E3 +419056.549}
SPL {X  -159.990, Y  +499.829, Z    +0.000, E1   +36.864, E3 +419073.354}
SPL {X  -159.990, Y  +498.054, Z    +0.000, E1   +35.692, E3 +419085.393}
ENDSPLINE

SPLINE
SPL {X  -159.990, Y  +506.994, Z    +0.000, E1   +30.162, E3 +419092.054}
ENDSPLINE

SPLINE
SPL {X  -159.990, Y  +502.084, Z    +0.000, E1   +31.057, E3 +419103.706}
SPL {X  -159.990, Y  +494.586, Z    +0.000, E1   +32.444, E3 +419120.309}
SPL {X  -159.990, Y  +486.073, Z    +0.000, E1   +33.960, E3 +419138.147}
SPL {X  -159.990, Y  +477.314, Z    +0.000, E1   +35.342, E3 +419156.325}
SPL {X  -159.990, Y  +471.459, Z    +0.000, E1   +35.779, E3 +419170.864}
SPL {X  -159.990, Y  +467.485, Z    +0.000, E1   +35.768, E3 +419182.594}
SPL {X  -159.990, Y  +462.739, Z    +0.000, E1   +35.799, E3 +419196.522}
SPL {X  -159.990, Y  +457.385, Z    +0.000, E1   +35.788, E3 +419212.305}
SPL {X  -159.990, Y  +452.637, Z    +0.000, E1   +35.783, E3 +419226.297}
SPL {X  -159.990, Y  +446.982, Z    +0.000, E1   +35.815, E3 +419242.899}
SPL {X  -159.990, Y  +442.593, Z    +0.000, E1   +35.759, E3 +419255.908}
SPL {X  -159.990, Y  +439.109, Z    +0.000, E1   +35.781, E3 +419266.125}
SPL {X  -159.990, Y  +434.400, Z    +0.000, E1   +35.789, E3 +419279.980}
SPL {X  -159.990, Y  +430.115, Z    +0.000, E1   +35.777, E3 +419292.597}
SPL {X  -159.990, Y  +426.641, Z    +0.000, E1   +35.769, E3 +419302.847}
SPL {X  -159.990, Y  +422.627, Z    +0.000, E1   +35.788, E3 +419314.645}
SPL {X  -159.990, Y  +417.866, Z    +0.000, E1   +35.788, E3 +419328.658}
SPL {X  -159.990, Y  +413.498, Z    +0.000, E1   +35.779, E3 +419341.540}
SPL {X  -159.990, Y  +408.600, Z    +0.000, E1   +35.802, E3 +419355.928}
SPL {X  -159.990, Y  +403.496, Z    +0.000, E1   +35.787, E3 +419370.983}
SPL {X  -159.990, Y  +398.606, Z    +0.000, E1   +35.794, E3 +419385.370}
SPL {X  -159.990, Y  +394.138, Z    +0.000, E1   +35.778, E3 +419398.553}
SPL {X  -159.990, Y  +390.065, Z    +0.000, E1   +35.780, E3 +419410.544}
SPL {X  -159.990, Y  +385.506, Z    +0.000, E1   +35.789, E3 +419423.949}
SPL {X  -159.976, Y  +380.359, Z    +0.000, E1   +35.797, E3 +419439.098}
SPL {X  -159.831, Y  +375.358, Z    +0.000, E1   +35.763, E3 +419453.988}
SPL {X  -159.613, Y  +371.527, Z    +0.000, E1   +35.709, E3 +419465.543}
SPL {X  -159.203, Y  +366.647, Z    +0.000, E1   +35.680, E3 +419480.276}
SPL {X  -158.715, Y  +362.338, Z    +0.000, E1   +35.547, E3 +419493.581}
SPL {X  -158.237, Y  +358.884, Z    +0.000, E1   +35.480, E3 +419504.238}
SPL {X  -157.724, Y  +355.670, Z    +0.000, E1   +35.371, E3 +419514.272}
SPL {X  -157.185, Y  +352.671, Z    +0.000, E1   +35.292, E3 +419523.651}
SPL {X  -156.582, Y  +349.653, Z    +0.000, E1   +35.175, E3 +419533.184}
SPL {X  -155.743, Y  +345.880, Z    +0.000, E1   +35.068, E3 +419545.112}
SPL {X  -154.759, Y  +341.925, Z    +0.000, E1   +34.868, E3 +419557.818}
SPL {X  -154.305, Y  +340.232, Z    +0.000, E1   +28.975, E3 +419611.647}
ENDSPLINE

SPLINE
SPL {X  -158.456, Y  +360.399, Z    +0.000, E1   +16.490, E3 +419648.466}
SPL {X  -159.553, Y  +370.677, Z    +0.000, E1   +10.576, E3 +419656.227}
SPL {X  -159.960, Y  +379.402, Z    +0.000, E1    +5.303, E3 +419660.247}
SPL {X  -159.990, Y  +385.983, Z    +0.000, E1    +0.882, E3 +419662.319}
SPL {X  -159.990, Y  +390.933, Z    +0.000, E1    -2.877, E3 +419663.767}
SPL {X  -159.990, Y  +396.375, Z    +0.000, E1    -7.538, E3 +419665.542}
SPL {X  -159.990, Y  +404.277, Z    +0.000, E1   -14.543, E3 +419669.205}
SPL {X  -159.990, Y  +423.101, Z    +0.000, E1   -27.351, E3 +419685.644}
SPL {X  -159.990, Y  +430.396, Z    +0.000, E1   -30.473, E3 +419694.897}
SPL {X  -159.990, Y  +447.483, Z    +0.000, E1   -34.518, E3 +419725.080}
SPL {X  -159.990, Y  +453.425, Z    +0.000, E1   -35.055, E3 +419739.762}
SPL {X  -159.990, Y  +457.209, Z    +0.000, E1   -35.039, E3 +419751.238}
SPL {X  -159.990, Y  +460.708, Z    +0.000, E1   -35.045, E3 +419761.820}
SPL {X  -159.990, Y  +465.240, Z    +0.000, E1   -35.066, E3 +419775.495}
SPL {X  -159.990, Y  +470.278, Z    +0.000, E1   -35.063, E3 +419790.729}
SPL {X  -159.990, Y  +474.610, Z    +0.000, E1   -35.053, E3 +419803.828}
SPL {X  -159.990, Y  +478.303, Z    +0.000, E1   -35.049, E3 +419815.000}
SPL {X  -159.990, Y  +482.537, Z    +0.000, E1   -35.066, E3 +419827.791}
SPL {X  -159.990, Y  +487.181, Z    +0.000, E1   -35.054, E3 +419841.874}
SPL {X  -159.990, Y  +490.807, Z    +0.000, E1   -35.036, E3 +419852.875}
SPL {X  -159.990, Y  +493.669, Z    +0.000, E1   -35.034, E3 +419861.555}
SPL {X  -159.990, Y  +497.072, Z    +0.000, E1   -35.040, E3 +419871.842}
SPL {X  -159.990, Y  +500.395, Z    +0.000, E1   -35.033, E3 +419881.905}
SPL {X  -159.990, Y  +502.996, Z    +0.000, E1   -35.034, E3 +419889.753}
SPL {X  -159.990, Y  +507.359, Z    +0.000, E1   -35.080, E3 +419902.882}
SPL {X  -159.990, Y  +512.562, Z    +0.000, E1   -35.055, E3 +419918.664}
SPL {X  -159.990, Y  +517.156, Z    +0.000, E1   -35.059, E3 +419932.545}
SPL {X  -159.990, Y  +521.637, Z    +0.000, E1   -35.056, E3 +419946.109}
SPL {X  -159.990, Y  +526.246, Z    +0.000, E1   -35.065, E3 +419960.012}
SPL {X  -159.990, Y  +530.289, Z    +0.000, E1   -35.044, E3 +419972.298}
SPL {X  -159.990, Y  +534.797, Z    +0.000, E1   -35.069, E3 +419985.899}
SPL {X  -159.990, Y  +538.710, Z    +0.000, E1   -35.033, E3 +419997.796}
SPL {X  -159.990, Y  +542.114, Z    +0.000, E1   -35.053, E3 +420008.048}
SPL {X  -159.990, Y  +545.724, Z    +0.000, E1   -35.043, E3 +420018.972}
SPL {X  -159.990, Y  +549.546, Z    +0.000, E1   -35.061, E3 +420030.496}
SPL {X  -159.990, Y  +552.868, Z    +0.000, E1   -35.047, E3 +420040.538}
SPL {X  -159.990, Y  +557.043, Z    +0.000, E1   -35.087, E3 +420053.076}
SPL {X  -159.990, Y  +561.808, Z    +0.000, E1   -35.066, E3 +420067.529}
SPL {X  -159.990, Y  +566.542, Z    +0.000, E1   -35.080, E3 +420081.829}
SPL {X  -159.990, Y  +570.261, Z    +0.000, E1   -35.046, E3 +420093.125}
SPL {X  -159.990, Y  +574.780, Z    +0.000, E1   -35.101, E3 +420106.705}
SPL {X  -159.990, Y  +579.185, Z    +0.000, E1   -35.047, E3 +420120.106}
SPL {X  -159.990, Y  +581.944, Z    +0.000, E1   -35.051, E3 +420128.444}
SPL {X  -159.990, Y  +585.414, Z    +0.000, E1   -35.059, E3 +420138.927}
SPL {X  -159.990, Y  +590.166, Z    +0.000, E1   -35.084, E3 +420153.255}
SPL {X  -159.990, Y  +594.231, Z    +0.000, E1   -35.047, E3 +420165.606}
SPL {X  -159.990, Y  +598.554, Z    +0.000, E1   -35.088, E3 +420178.613}
SPL {X  -159.990, Y  +602.221, Z    +0.000, E1   -35.048, E3 +420189.744}
SPL {X  -159.990, Y  +605.846, Z    +0.000, E1   -35.077, E3 +420200.668}
SPL {X  -159.990, Y  +609.372, Z    +0.000, E1   -35.047, E3 +420211.365}
SPL {X  -159.990, Y  +613.036, Z    +0.000, E1   -35.082, E3 +420222.400}
SPL {X  -159.990, Y  +617.577, Z    +0.000, E1   -35.061, E3 +420236.162}
SPL {X  -159.990, Y  +621.534, Z    +0.000, E1   -35.068, E3 +420248.096}
SPL {X  -159.990, Y  +626.426, Z    +0.000, E1   -35.093, E3 +420262.855}
SPL {X  -159.990, Y  +631.553, Z    +0.000, E1   -35.068, E3 +420278.413}
SPL {X  -159.990, Y  +635.965, Z    +0.000, E1   -35.065, E3 +420291.762}
SPL {X  -159.990, Y  +640.633, Z    +0.000, E1   -35.080, E3 +420305.850}
SPL {X  -159.990, Y  +645.423, Z    +0.000, E1   -35.070, E3 +420320.355}
SPL {X  -159.990, Y  +650.555, Z    +0.000, E1   -35.089, E3 +420335.845}
SPL {X  -159.990, Y  +656.270, Z    +0.000, E1   -35.087, E3 +420353.137}
SPL {X  -159.990, Y  +661.105, Z    +0.000, E1   -35.059, E3 +420367.801}
SPL {X  -159.990, Y  +665.311, Z    +0.000, E1   -35.064, E3 +420380.516}
SPL {X  -159.990, Y  +668.650, Z    +0.000, E1   -35.040, E3 +420390.655}
SPL {X  -159.990, Y  +671.288, Z    +0.000, E1   -35.046, E3 +420398.620}
SPL {X  -159.948, Y  +675.148, Z    +0.000, E1   -35.069, E3 +420410.255}
SPL {X  -159.752, Y  +680.228, Z    +0.000, E1   -35.050, E3 +420425.803}
SPL {X  -159.371, Y  +685.563, Z    +0.000, E1   -34.989, E3 +420442.314}
SPL {X  -158.886, Y  +690.264, Z    +0.000, E1   -34.888, E3 +420457.066}
SPL {X  -158.362, Y  +694.266, Z    +0.000, E1   -34.794, E3 +420469.739}
SPL {X  -157.614, Y  +698.973, Z    +0.000, E1   -34.690, E3 +420484.740}
SPL {X  -156.901, Y  +702.787, Z    +0.000, E1   -34.523, E3 +420497.083}
SPL {X  -156.097, Y  +706.580, Z    +0.000, E1   -34.427, E3 +420509.323}
SPL {X  -155.080, Y  +710.833, Z    +0.000, E1   -34.231, E3 +420523.257}
SPL {X  -153.949, Y  +715.047, Z    +0.000, E1   -29.578, E3 +420576.807}
ENDSPLINE

SPLINE
SPL {X  -158.529, Y  +693.075, Z    +0.000, E1   -15.996, E3 +420620.792}
SPL {X  -159.750, Y  +680.262, Z    +0.000, E1    -8.563, E3 +420629.203}
SPL {X  -159.973, Y  +673.798, Z    +0.000, E1    -4.600, E3 +420631.667}
SPL {X  -159.990, Y  +668.863, Z    +0.000, E1    -1.298, E3 +420633.106}
SPL {X  -159.990, Y  +663.839, Z    +0.000, E1    +2.454, E3 +420634.367}
SPL {X  -159.990, Y  +658.349, Z    +0.000, E1    +7.223, E3 +420636.049}
SPL {X  -159.990, Y  +650.390, Z    +0.000, E1   +14.372, E3 +420639.795}
SPL {X  -159.990, Y  +643.417, Z    +0.000, E1   +20.300, E3 +420644.059}
SPL {X  -159.990, Y  +621.124, Z    +0.000, E1   +32.598, E3 +420665.773}
SPL {X  -159.990, Y  +597.855, Z    +0.000, E1   +36.862, E3 +420708.692}
SPL {X  -159.990, Y  +593.971, Z    +0.000, E1   +36.841, E3 +420719.724}
SPL {X  -159.990, Y  +589.749, Z    +0.000, E1   +36.860, E3 +420731.651}
SPL {X  -159.990, Y  +585.754, Z    +0.000, E1   +36.838, E3 +420743.006}
SPL {X  -159.990, Y  +581.795, Z    +0.000, E1   +36.847, E3 +420754.219}
SPL {X  -159.990, Y  +577.286, Z    +0.000, E1   +36.853, E3 +420766.976}
SPL {X  -159.990, Y  +572.409, Z    +0.000, E1   +36.854, E3 +420780.788}
SPL {X  -159.990, Y  +567.110, Z    +0.000, E1   +36.868, E3 +420795.749}
SPL {X  -159.990, Y  +562.387, Z    +0.000, E1   +36.853, E3 +420809.110}
SPL {X  -159.990, Y  +557.944, Z    +0.000, E1   +36.859, E3 +420821.704}
SPL {X  -159.990, Y  +553.661, Z    +0.000, E1   +36.844, E3 +420833.868}
SPL {X  -159.990, Y  +549.195, Z    +0.000, E1   +36.856, E3 +420846.503}
SPL {X  -159.990, Y  +544.733, Z    +0.000, E1   +36.845, E3 +420859.149}
SPL {X  -159.990, Y  +539.889, Z    +0.000, E1   +36.872, E3 +420872.833}
SPL {X  -159.990, Y  +534.469, Z    +0.000, E1   +36.855, E3 +420888.231}
SPL {X  -159.990, Y  +528.569, Z    +0.000, E1   +36.871, E3 +420904.949}
SPL {X  -159.990, Y  +522.641, Z    +0.000, E1   +36.854, E3 +420921.760}
SPL {X  -159.990, Y  +517.225, Z    +0.000, E1   +36.859, E3 +420937.094}
SPL {X  -159.990, Y  +511.408, Z    +0.000, E1   +36.858, E3 +420953.582}
SPL {X  -159.990, Y  +507.404, Z    +0.000, E1   +36.819, E3 +420964.985}
SPL {X  -159.990, Y  +503.454, Z    +0.000, E1   +36.847, E3 +420976.139}
SPL {X  -159.990, Y  +498.507, Z    +0.000, E1   +36.487, E3 +420992.588}
ENDSPLINE

SPLINE
SPL {X  -159.990, Y  +505.140, Z    +0.000, E1   +30.523, E3 +421009.463}
ENDSPLINE

SPLINE
SPL {X  -159.990, Y  +497.800, Z    +0.000, E1   +31.845, E3 +421026.419}
SPL {X  -159.990, Y  +489.306, Z    +0.000, E1   +33.397, E3 +421044.498}
SPL {X  -159.990, Y  +481.374, Z    +0.000, E1   +34.706, E3 +421061.009}
SPL {X  -159.990, Y  +475.503, Z    +0.000, E1   +35.597, E3 +421073.062}
SPL {X  -159.990, Y  +471.459, Z    +0.000, E1   +35.779, E3 +421083.908}
SPL {X  -159.990, Y  +466.474, Z    +0.000, E1   +35.796, E3 +421098.567}
SPL {X  -159.990, Y  +461.990, Z    +0.000, E1   +35.776, E3 +421111.802}
SPL {X  -159.990, Y  +458.524, Z    +0.000, E1   +35.761, E3 +421122.039}
SPL {X  -159.990, Y  +453.597, Z    +0.000, E1   +35.819, E3 +421136.459}
SPL {X  -159.990, Y  +448.227, Z    +0.000, E1   +35.776, E3 +421152.337}
SPL {X  -159.990, Y  +443.707, Z    +0.000, E1   +35.784, E3 +421165.633}
SPL {X  -159.990, Y  +439.109, Z    +0.000, E1   +35.781, E3 +421179.169}
SPL {X  -159.990, Y  +435.535, Z    +0.000, E1   +35.764, E3 +421189.719}
SPL {X  -159.990, Y  +431.100, Z    +0.000, E1   +35.807, E3 +421202.704}
SPL {X  -159.990, Y  +425.407, Z    +0.000, E1   +35.800, E3 +421219.480}
SPL {X  -159.990, Y  +420.199, Z    +0.000, E1   +35.790, E3 +421234.834}
SPL {X  -159.990, Y  +414.514, Z    +0.000, E1   +35.815, E3 +421251.533}
SPL {X  -159.990, Y  +408.600, Z    +0.000, E1   +35.802, E3 +421268.971}
SPL {X  -159.990, Y  +403.496, Z    +0.000, E1   +35.787, E3 +421284.026}
SPL {X  -159.990, Y  +398.606, Z    +0.000, E1   +35.794, E3 +421298.414}
SPL {X  -159.990, Y  +394.138, Z    +0.000, E1   +35.778, E3 +421311.597}
SPL {X  -159.990, Y  +388.813, Z    +0.000, E1   +35.819, E3 +421327.209}
SPL {X  -159.990, Y  +383.172, Z    +0.000, E1   +35.789, E3 +421343.863}
SPL {X  -159.936, Y  +378.352, Z    +0.000, E1   +35.782, E3 +421358.102}
SPL {X  -159.693, Y  +372.749, Z    +0.000, E1   +35.767, E3 +421374.834}
SPL {X  -159.203, Y  +366.647, Z    +0.000, E1   +35.680, E3 +421393.320}
SPL {X  -158.715, Y  +362.338, Z    +0.000, E1   +35.547, E3 +421406.625}
SPL {X  -158.237, Y  +358.884, Z    +0.000, E1   +35.480, E3 +421417.282}
SPL {X  -157.724, Y  +355.670, Z    +0.000, E1   +35.371, E3 +421427.316}
SPL {X  -157.185, Y  +352.671, Z    +0.000, E1   +35.292, E3 +421436.695}
SPL {X  -156.302, Y  +348.345, Z    +0.000, E1   +35.165, E3 +421450.316}
SPL {X  -155.054, Y  +343.066, Z    +0.000, E1   +34.964, E3 +421467.130}
SPL {X  -154.305, Y  +340.232, Z    +0.000, E1   +28.975, E3 +421524.690}
ENDSPLINE

SPLINE
SPL {X  -158.456, Y  +360.399, Z    +0.000, E1   +16.490, E3 +421561.510}
SPL {X  -159.553, Y  +370.677, Z    +0.000, E1   +10.576, E3 +421569.270}
SPL {X  -159.960, Y  +379.402, Z    +0.000, E1    +5.303, E3 +421573.290}
SPL {X  -159.990, Y  +387.301, Z    +0.000, E1    +0.001, E3 +421575.752}
SPL {X  -159.990, Y  +392.161, Z    +0.000, E1    -3.946, E3 +421577.163}
SPL {X  -159.990, Y  +396.375, Z    +0.000, E1    -7.538, E3 +421578.585}
SPL {X  -159.990, Y  +404.277, Z    +0.000, E1   -14.543, E3 +421582.248}
SPL {X  -159.990, Y  +423.101, Z    +0.000, E1   -27.351, E3 +421598.687}
SPL {X  -159.990, Y  +430.933, Z    +0.000, E1   -30.672, E3 +421608.658}
SPL {X  -159.990, Y  +452.779, Z    +0.000, E1   -35.077, E3 +421650.821}
SPL {X  -159.990, Y  +457.209, Z    +0.000, E1   -35.039, E3 +421664.281}
SPL {X  -159.990, Y  +460.708, Z    +0.000, E1   -35.045, E3 +421674.863}
SPL {X  -159.990, Y  +464.162, Z    +0.000, E1   -35.038, E3 +421685.320}
SPL {X  -159.990, Y  +467.857, Z    +0.000, E1   -35.053, E3 +421696.477}
SPL {X  -159.990, Y  +471.326, Z    +0.000, E1   -35.038, E3 +421706.972}
SPL {X  -159.990, Y  +474.610, Z    +0.000, E1   -35.053, E3 +421716.871}
SPL {X  -159.990, Y  +479.424, Z    +0.000, E1   -35.081, E3 +421731.383}
SPL {X  -159.990, Y  +483.513, Z    +0.000, E1   -35.038, E3 +421743.837}
SPL {X  -159.990, Y  +487.181, Z    +0.000, E1   -35.054, E3 +421754.917}
SPL {X  -159.990, Y  +492.368, Z    +0.000, E1   -35.076, E3 +421770.589}
SPL {X  -159.990, Y  +497.072, Z    +0.000, E1   -35.040, E3 +421784.886}
SPL {X  -159.990, Y  +501.645, Z    +0.000, E1   -35.067, E3 +421798.669}
SPL {X  -159.990, Y  +506.307, Z    +0.000, E1   -35.049, E3 +421812.791}
SPL {X  -159.990, Y  +510.443, Z    +0.000, E1   -35.051, E3 +421825.303}
SPL {X  -159.990, Y  +514.632, Z    +0.000, E1   -35.050, E3 +421837.973}
SPL {X  -159.990, Y  +518.055, Z    +0.000, E1   -35.037, E3 +421848.342}
SPL {X  -159.990, Y  +521.637, Z    +0.000, E1   -35.056, E3 +421859.152}
SPL {X  -159.990, Y  +525.227, Z    +0.000, E1   -35.041, E3 +421870.013}
SPL {X  -159.990, Y  +529.413, Z    +0.000, E1   -35.072, E3 +421882.642}
SPL {X  -159.990, Y  +533.060, Z    +0.000, E1   -35.029, E3 +421893.748}
SPL {X  -159.990, Y  +537.053, Z    +0.000, E1   -35.083, E3 +421905.744}
SPL {X  -159.990, Y  +542.114, Z    +0.000, E1   -35.053, E3 +421921.091}
SPL {X  -159.990, Y  +545.724, Z    +0.000, E1   -35.043, E3 +421932.016}
SPL {X  -159.990, Y  +549.546, Z    +0.000, E1   -35.061, E3 +421943.540}
SPL {X  -159.990, Y  +552.868, Z    +0.000, E1   -35.047, E3 +421953.582}
SPL {X  -159.990, Y  +557.043, Z    +0.000, E1   -35.087, E3 +421966.119}
SPL {X  -159.990, Y  +561.808, Z    +0.000, E1   -35.066, E3 +421980.572}
SPL {X  -159.990, Y  +566.542, Z    +0.000, E1   -35.080, E3 +421994.873}
SPL {X  -159.990, Y  +571.374, Z    +0.000, E1   -35.070, E3 +422009.496}
SPL {X  -159.990, Y  +575.771, Z    +0.000, E1   -35.064, E3 +422022.802}
SPL {X  -159.990, Y  +580.750, Z    +0.000, E1   -35.087, E3 +422037.824}
SPL {X  -159.990, Y  +585.414, Z    +0.000, E1   -35.059, E3 +422051.970}
SPL {X  -159.990, Y  +590.166, Z    +0.000, E1   -35.084, E3 +422066.299}
SPL {X  -159.990, Y  +594.231, Z    +0.000, E1   -35.047, E3 +422078.650}
SPL {X  -159.990, Y  +598.554, Z    +0.000, E1   -35.088, E3 +422091.656}
SPL {X  -159.990, Y  +603.289, Z    +0.000, E1   -35.068, E3 +422105.984}
SPL {X  -159.990, Y  +607.919, Z    +0.000, E1   -35.079, E3 +422119.973}
SPL {X  -159.990, Y  +612.068, Z    +0.000, E1   -35.057, E3 +422132.553}
SPL {X  -159.990, Y  +616.690, Z    +0.000, E1   -35.089, E3 +422146.480}
SPL {X  -159.990, Y  +621.534, Z    +0.000, E1   -35.068, E3 +422161.139}
SPL {X  -159.990, Y  +625.237, Z    +0.000, E1   -35.062, E3 +422172.341}
SPL {X  -159.990, Y  +629.217, Z    +0.000, E1   -35.065, E3 +422184.399}
SPL {X  -159.990, Y  +632.566, Z    +0.000, E1   -35.044, E3 +422194.561}
SPL {X  -159.990, Y  +636.917, Z    +0.000, E1   -35.095, E3 +422207.636}
SPL {X  -159.990, Y  +641.534, Z    +0.000, E1   -35.053, E3 +422221.663}
SPL {X  -159.990, Y  +645.423, Z    +0.000, E1   -35.070, E3 +422233.399}
SPL {X  -159.990, Y  +650.555, Z    +0.000, E1   -35.089, E3 +422248.888}
SPL {X  -159.990, Y  +654.793, Z    +0.000, E1   -35.049, E3 +422261.768}
SPL {X  -159.990, Y  +657.535, Z    +0.000, E1   -35.049, E3 +422270.064}
SPL {X  -159.990, Y  +661.105, Z    +0.000, E1   -35.059, E3 +422280.845}
SPL {X  -159.990, Y  +665.311, Z    +0.000, E1   -35.064, E3 +422293.559}
SPL {X  -159.990, Y  +670.193, Z    +0.000, E1   -35.076, E3 +422308.306}
SPL {X  -159.948, Y  +675.148, Z    +0.000, E1   -35.069, E3 +422323.299}
SPL {X  -159.752, Y  +680.228, Z    +0.000, E1   -35.050, E3 +422338.846}
SPL {X  -159.371, Y  +685.563, Z    +0.000, E1   -34.989, E3 +422355.358}
SPL {X  -158.886, Y  +690.264, Z    +0.000, E1   -34.888, E3 +422370.109}
SPL {X  -158.362, Y  +694.266, Z    +0.000, E1   -34.794, E3 +422382.783}
SPL {X  -157.614, Y  +698.973, Z    +0.000, E1   -34.690, E3 +422397.783}
SPL {X  -156.640, Y  +704.066, Z    +0.000, E1   -34.516, E3 +422414.208}
SPL {X  -155.835, Y  +707.723, Z    +0.000, E1   -34.344, E3 +422426.151}
SPL {X  -155.153, Y  +710.542, Z    +0.000, E1   -34.234, E3 +422435.370}
SPL {X  -153.767, Y  +715.686, Z    +0.000, E1   -30.747, E3 +422480.588}
ENDSPLINE

SPLINE
SPL {X  -154.589, Y  +712.719, Z    +0.000, E1   -27.400, E3 +422501.988}
SPL {X  -158.529, Y  +693.075, Z    +0.000, E1   -15.996, E3 +422533.835}
SPL {X  -159.750, Y  +680.262, Z    +0.000, E1    -8.563, E3 +422542.246}
SPL {X  -159.973, Y  +673.798, Z    +0.000, E1    -4.600, E3 +422544.710}
SPL {X  -159.990, Y  +667.448, Z    +0.000, E1    -0.356, E3 +422546.490}
SPL {X  -159.990, Y  +662.686, Z    +0.000, E1    +3.472, E3 +422547.725}
SPL {X  -159.990, Y  +658.349, Z    +0.000, E1    +7.223, E3 +422549.093}
SPL {X  -159.990, Y  +653.910, Z    +0.000, E1   +11.344, E3 +422550.860}
SPL {X  -159.990, Y  +646.193, Z    +0.000, E1   +17.980, E3 +422555.330}
SPL {X  -159.990, Y  +621.124, Z    +0.000, E1   +32.598, E3 +422578.816}
SPL {X  -159.990, Y  +599.888, Z    +0.000, E1   +36.828, E3 +422616.056}
SPL {X  -159.990, Y  +595.346, Z    +0.000, E1   +36.880, E3 +422628.822}
SPL {X  -159.990, Y  +589.749, Z    +0.000, E1   +36.860, E3 +422644.695}
SPL {X  -159.990, Y  +585.754, Z    +0.000, E1   +36.838, E3 +422656.050}
SPL {X  -159.990, Y  +581.795, Z    +0.000, E1   +36.847, E3 +422667.262}
SPL {X  -159.990, Y  +576.165, Z    +0.000, E1   +36.887, E3 +422683.142}
SPL {X  -159.990, Y  +570.328, Z    +0.000, E1   +36.855, E3 +422699.715}
SPL {X  -159.990, Y  +566.126, Z    +0.000, E1   +36.841, E3 +422711.621}
SPL {X  -159.990, Y  +562.387, Z    +0.000, E1   +36.853, E3 +422722.154}
SPL {X  -159.990, Y  +557.944, Z    +0.000, E1   +36.859, E3 +422734.748}
SPL {X  -159.990, Y  +552.571, Z    +0.000, E1   +36.873, E3 +422749.952}
SPL {X  -159.990, Y  +548.223, Z    +0.000, E1   +36.832, E3 +422762.342}
SPL {X  -159.990, Y  +543.458, Z    +0.000, E1   +36.882, E3 +422775.745}
SPL {X  -159.990, Y  +537.639, Z    +0.000, E1   +36.860, E3 +422792.283}
SPL {X  -159.990, Y  +531.894, Z    +0.000, E1   +36.865, E3 +422808.572}
SPL {X  -159.990, Y  +525.940, Z    +0.000, E1   +36.859, E3 +422825.454}
SPL {X  -159.990, Y  +520.301, Z    +0.000, E1   +36.855, E3 +422841.431}
SPL {X  -159.990, Y  +516.005, Z    +0.000, E1   +36.824, E3 +422853.657}
SPL {X  -159.990, Y  +511.408, Z    +0.000, E1   +36.858, E3 +422866.626}
SPL {X  -159.990, Y  +505.756, Z    +0.000, E1   +36.857, E3 +422882.636}
SPL {X  -159.990, Y  +499.829, Z    +0.000, E1   +36.864, E3 +422899.440}
SPL {X  -159.990, Y  +498.054, Z    +0.000, E1   +35.692, E3 +422911.480}
ENDSPLINE

SPLINE
SPL {X  -159.990, Y  +506.994, Z    +0.000, E1   +30.162, E3 +422918.141}
ENDSPLINE

SPLINE
SPL {X  -159.990, Y  +502.084, Z    +0.000, E1   +31.057, E3 +422929.793}
SPL {X  -159.990, Y  +494.586, Z    +0.000, E1   +32.444, E3 +422946.396}
SPL {X  -159.990, Y  +487.723, Z    +0.000, E1   +33.658, E3 +422960.849}
SPL {X  -159.990, Y  +481.374, Z    +0.000, E1   +34.706, E3 +422974.052}
SPL {X  -159.990, Y  +475.503, Z    +0.000, E1   +35.597, E3 +422986.105}
SPL {X  -159.990, Y  +471.459, Z    +0.000, E1   +35.779, E3 +422996.951}
SPL {X  -159.990, Y  +466.474, Z    +0.000, E1   +35.796, E3 +423011.610}
SPL {X  -159.990, Y  +461.990, Z    +0.000, E1   +35.776, E3 +423024.846}
SPL {X  -159.990, Y  +457.385, Z    +0.000, E1   +35.788, E3 +423038.392}
SPL {X  -159.990, Y  +452.637, Z    +0.000, E1   +35.783, E3 +423052.384}
SPL {X  -159.990, Y  +446.982, Z    +0.000, E1   +35.815, E3 +423068.986}
SPL {X  -159.990, Y  +442.593, Z    +0.000, E1   +35.759, E3 +423081.995}
SPL {X  -159.990, Y  +439.109, Z    +0.000, E1   +35.781, E3 +423092.212}
SPL {X  -159.990, Y  +435.535, Z    +0.000, E1   +35.764, E3 +423102.763}
SPL {X  -159.990, Y  +431.100, Z    +0.000, E1   +35.807, E3 +423115.748}
SPL {X  -159.990, Y  +426.641, Z    +0.000, E1   +35.769, E3 +423128.934}
SPL {X  -159.990, Y  +422.627, Z    +0.000, E1   +35.788, E3 +423140.732}
SPL {X  -159.990, Y  +417.866, Z    +0.000, E1   +35.788, E3 +423154.745}
SPL {X  -159.990, Y  +413.498, Z    +0.000, E1   +35.779, E3 +423167.627}
SPL {X  -159.990, Y  +408.600, Z    +0.000, E1   +35.802, E3 +423182.015}
SPL {X  -159.990, Y  +403.496, Z    +0.000, E1   +35.787, E3 +423197.070}
SPL {X  -159.990, Y  +398.606, Z    +0.000, E1   +35.794, E3 +423211.457}
SPL {X  -159.990, Y  +394.138, Z    +0.000, E1   +35.778, E3 +423224.640}
SPL {X  -159.990, Y  +388.813, Z    +0.000, E1   +35.819, E3 +423240.252}
SPL {X  -159.990, Y  +383.172, Z    +0.000, E1   +35.789, E3 +423256.906}
SPL {X  -159.936, Y  +378.352, Z    +0.000, E1   +35.782, E3 +423271.145}
SPL {X  -159.790, Y  +374.497, Z    +0.000, E1   +35.735, E3 +423282.690}
SPL {X  -159.547, Y  +370.604, Z    +0.000, E1   +35.724, E3 +423294.375}
SPL {X  -159.134, Y  +365.969, Z    +0.000, E1   +35.644, E3 +423308.460}
SPL {X  -158.715, Y  +362.338, Z    +0.000, E1   +35.547, E3 +423319.668}
SPL {X  -158.237, Y  +358.884, Z    +0.000, E1   +35.480, E3 +423330.325}
SPL {X  -157.724, Y  +355.670, Z    +0.000, E1   +35.371, E3 +423340.359}
SPL {X  -157.185, Y  +352.671, Z    +0.000, E1   +35.292, E3 +423349.738}
SPL {X  -156.582, Y  +349.653, Z    +0.000, E1   +35.175, E3 +423359.271}
SPL {X  -155.743, Y  +345.880, Z    +0.000, E1   +35.068, E3 +423371.198}
SPL {X  -154.759, Y  +341.925, Z    +0.000, E1   +34.868, E3 +423383.905}
SPL {X  -154.305, Y  +340.232, Z    +0.000, E1   +28.975, E3 +423437.734}
ENDSPLINE

SPLINE
SPL {X  -158.456, Y  +360.399, Z    +0.000, E1   +16.490, E3 +423474.553}
SPL {X  -159.553, Y  +370.677, Z    +0.000, E1   +10.576, E3 +423482.314}
SPL {X  -159.960, Y  +379.402, Z    +0.000, E1    +5.303, E3 +423486.334}
SPL {X  -159.990, Y  +385.983, Z    +0.000, E1    +0.882, E3 +423488.406}
SPL {X  -159.990, Y  +390.933, Z    +0.000, E1    -2.877, E3 +423489.854}
SPL {X  -159.990, Y  +396.375, Z    +0.000, E1    -7.538, E3 +423491.629}
SPL {X  -159.990, Y  +404.277, Z    +0.000, E1   -14.543, E3 +423495.292}
SPL {X  -159.990, Y  +423.101, Z    +0.000, E1   -27.351, E3 +423511.731}
SPL {X  -159.990, Y  +430.933, Z    +0.000, E1   -30.672, E3 +423521.702}
SPL {X  -159.990, Y  +452.779, Z    +0.000, E1   -35.077, E3 +423563.865}
SPL {X  -159.990, Y  +457.209, Z    +0.000, E1   -35.039, E3 +423577.324}
SPL {X  -159.990, Y  +460.708, Z    +0.000, E1   -35.045, E3 +423587.907}
SPL {X  -159.990, Y  +464.162, Z    +0.000, E1   -35.038, E3 +423598.363}
SPL {X  -159.990, Y  +467.857, Z    +0.000, E1   -35.053, E3 +423609.520}
SPL {X  -159.990, Y  +471.326, Z    +0.000, E1   -35.038, E3 +423620.015}
SPL {X  -159.990, Y  +474.610, Z    +0.000, E1   -35.053, E3 +423629.915}
SPL {X  -159.990, Y  +478.303, Z    +0.000, E1   -35.049, E3 +423641.087}
SPL {X  -159.990, Y  +482.537, Z    +0.000, E1   -35.066, E3 +423653.878}
SPL {X  -159.990, Y  +487.181, Z    +0.000, E1   -35.054, E3 +423667.961}
SPL {X  -159.990, Y  +492.368, Z    +0.000, E1   -35.076, E3 +423683.633}
SPL {X  -159.990, Y  +497.072, Z    +0.000, E1   -35.040, E3 +423697.929}
SPL {X  -159.990, Y  +501.645, Z    +0.000, E1   -35.067, E3 +423711.712}
SPL {X  -159.990, Y  +506.307, Z    +0.000, E1   -35.049, E3 +423725.834}
SPL {X  -159.990, Y  +510.443, Z    +0.000, E1   -35.051, E3 +423738.347}
SPL {X  -159.990, Y  +514.632, Z    +0.000, E1   -35.050, E3 +423751.017}
SPL {X  -159.990, Y  +518.055, Z    +0.000, E1   -35.037, E3 +423761.386}
SPL {X  -159.990, Y  +521.637, Z    +0.000, E1   -35.056, E3 +423772.196}
SPL {X  -159.990, Y  +526.246, Z    +0.000, E1   -35.065, E3 +423786.099}
SPL {X  -159.990, Y  +531.319, Z    +0.000, E1   -35.072, E3 +423801.455}
SPL {X  -159.990, Y  +537.053, Z    +0.000, E1   -35.083, E3 +423818.788}
SPL {X  -159.990, Y  +542.114, Z    +0.000, E1   -35.053, E3 +423834.135}
SPL {X  -159.990, Y  +545.724, Z    +0.000, E1   -35.043, E3 +423845.059}
SPL {X  -159.990, Y  +549.546, Z    +0.000, E1   -35.061, E3 +423856.583}
SPL {X  -159.990, Y  +552.868, Z    +0.000, E1   -35.047, E3 +423866.625}
SPL {X  -159.990, Y  +557.043, Z    +0.000, E1   -35.087, E3 +423879.163}
SPL {X  -159.990, Y  +562.842, Z    +0.000, E1   -35.098, E3 +423896.696}
SPL {X  -159.990, Y  +568.750, Z    +0.000, E1   -35.087, E3 +423914.581}
SPL {X  -159.990, Y  +574.780, Z    +0.000, E1   -35.101, E3 +423932.792}
SPL {X  -159.990, Y  +580.750, Z    +0.000, E1   -35.087, E3 +423950.867}
SPL {X  -159.990, Y  +585.414, Z    +0.000, E1   -35.059, E3 +423965.014}
SPL {X  -159.990, Y  +588.716, Z    +0.000, E1   -35.047, E3 +423975.017}
SPL {X  -159.990, Y  +591.475, Z    +0.000, E1   -35.047, E3 +423983.357}
SPL {X  -159.990, Y  +595.313, Z    +0.000, E1   -35.073, E3 +423994.921}
SPL {X  -159.990, Y  +600.543, Z    +0.000, E1   -35.091, E3 +424010.703}
SPL {X  -159.990, Y  +605.846, Z    +0.000, E1   -35.077, E3 +424026.754}
SPL {X  -159.990, Y  +609.372, Z    +0.000, E1   -35.047, E3 +424037.452}
SPL {X  -159.990, Y  +613.036, Z    +0.000, E1   -35.082, E3 +424048.487}
SPL {X  -159.990, Y  +617.577, Z    +0.000, E1   -35.061, E3 +424062.249}
SPL {X  -159.990, Y  +621.534, Z    +0.000, E1   -35.068, E3 +424074.183}
SPL {X  -159.990, Y  +625.237, Z    +0.000, E1   -35.062, E3 +424085.385}
SPL {X  -159.990, Y  +629.217, Z    +0.000, E1   -35.065, E3 +424097.442}
SPL {X  -159.990, Y  +632.566, Z    +0.000, E1   -35.044, E3 +424107.605}
SPL {X  -159.990, Y  +636.917, Z    +0.000, E1   -35.095, E3 +424120.679}
SPL {X  -159.990, Y  +641.534, Z    +0.000, E1   -35.053, E3 +424134.707}
SPL {X  -159.990, Y  +645.423, Z    +0.000, E1   -35.070, E3 +424146.442}
SPL {X  -159.990, Y  +650.555, Z    +0.000, E1   -35.089, E3 +424161.932}
SPL {X  -159.990, Y  +656.270, Z    +0.000, E1   -35.087, E3 +424179.224}
SPL {X  -159.990, Y  +661.105, Z    +0.000, E1   -35.059, E3 +424193.888}
SPL {X  -159.990, Y  +665.311, Z    +0.000, E1   -35.064, E3 +424206.603}
SPL {X  -159.990, Y  +670.193, Z    +0.000, E1   -35.076, E3 +424221.350}
SPL {X  -159.948, Y  +675.148, Z    +0.000, E1   -35.069, E3 +424236.342}
SPL {X  -159.752, Y  +680.228, Z    +0.000, E1   -35.050, E3 +424251.890}
SPL {X  -159.371, Y  +685.563, Z    +0.000, E1   -34.989, E3 +424268.401}
SPL {X  -158.886, Y  +690.264, Z    +0.000, E1   -34.888, E3 +424283.153}
SPL {X  -158.362, Y  +694.266, Z    +0.000, E1   -34.794, E3 +424295.826}
SPL {X  -157.614, Y  +698.973, Z    +0.000, E1   -34.690, E3 +424310.827}
SPL {X  -156.640, Y  +704.066, Z    +0.000, E1   -34.516, E3 +424327.252}
SPL {X  -155.835, Y  +707.723, Z    +0.000, E1   -34.344, E3 +424339.194}
SPL {X  -155.080, Y  +710.833, Z    +0.000, E1   -34.231, E3 +424349.344}
SPL {X  -153.949, Y  +715.047, Z    +0.000, E1   -29.578, E3 +424402.894}
ENDSPLINE

SPLINE
SPL {X  -158.529, Y  +693.075, Z    +0.000, E1   -15.996, E3 +424446.879}
SPL {X  -159.750, Y  +680.262, Z    +0.000, E1    -8.563, E3 +424455.290}
SPL {X  -159.973, Y  +673.798, Z    +0.000, E1    -4.600, E3 +424457.754}
SPL {X  -159.990, Y  +668.863, Z    +0.000, E1    -1.298, E3 +424459.193}
SPL {X  -159.990, Y  +663.839, Z    +0.000, E1    +2.454, E3 +424460.454}
SPL {X  -159.990, Y  +658.349, Z    +0.000, E1    +7.223, E3 +424462.136}
SPL {X  -159.990, Y  +650.390, Z    +0.000, E1   +14.372, E3 +424465.882}
SPL {X  -159.990, Y  +643.417, Z    +0.000, E1   +20.300, E3 +424470.146}
SPL {X  -159.990, Y  +621.124, Z    +0.000, E1   +32.598, E3 +424491.860}
SPL {X  -159.990, Y  +597.855, Z    +0.000, E1   +36.862, E3 +424534.779}
SPL {X  -159.990, Y  +593.971, Z    +0.000, E1   +36.841, E3 +424545.811}
SPL {X  -159.990, Y  +589.749, Z    +0.000, E1   +36.860, E3 +424557.738}
SPL {X  -159.990, Y  +585.754, Z    +0.000, E1   +36.838, E3 +424569.093}
SPL {X  -159.990, Y  +581.795, Z    +0.000, E1   +36.847, E3 +424580.306}
SPL {X  -159.990, Y  +577.286, Z    +0.000, E1   +36.853, E3 +424593.062}
SPL {X  -159.990, Y  +572.409, Z    +0.000, E1   +36.854, E3 +424606.875}
SPL {X  -159.990, Y  +567.110, Z    +0.000, E1   +36.868, E3 +424621.836}
SPL {X  -159.990, Y  +562.387, Z    +0.000, E1   +36.853, E3 +424635.197}
SPL {X  -159.990, Y  +557.944, Z    +0.000, E1   +36.859, E3 +424647.791}
SPL {X  -159.990, Y  +553.661, Z    +0.000, E1   +36.844, E3 +424659.955}
SPL {X  -159.990, Y  +549.195, Z    +0.000, E1   +36.856, E3 +424672.590}
SPL {X  -159.990, Y  +544.733, Z    +0.000, E1   +36.845, E3 +424685.236}
SPL {X  -159.990, Y  +539.889, Z    +0.000, E1   +36.872, E3 +424698.920}
SPL {X  -159.990, Y  +534.469, Z    +0.000, E1   +36.855, E3 +424714.318}
SPL {X  -159.990, Y  +530.428, Z    +0.000, E1   +36.821, E3 +424725.852}
SPL {X  -159.990, Y  +525.940, Z    +0.000, E1   +36.859, E3 +424738.498}
SPL {X  -159.990, Y  +520.301, Z    +0.000, E1   +36.855, E3 +424754.474}
SPL {X  -159.990, Y  +516.005, Z    +0.000, E1   +36.824, E3 +424766.701}
SPL {X  -159.990, Y  +511.408, Z    +0.000, E1   +36.858, E3 +424779.669}
SPL {X  -159.990, Y  +505.756, Z    +0.000, E1   +36.857, E3 +424795.679}
SPL {X  -159.990, Y  +499.829, Z    +0.000, E1   +36.864, E3 +424812.484}
SPL {X  -159.990, Y  +498.054, Z    +0.000, E1   +35.692, E3 +424824.523}
ENDSPLINE

SPLINE
SPL {X  -159.990, Y  +505.140, Z    +0.000, E1   +30.523, E3 +424835.550}
ENDSPLINE

SPLINE
SPL {X  -159.990, Y  +497.800, Z    +0.000, E1   +31.845, E3 +424852.506}
SPL {X  -159.990, Y  +492.180, Z    +0.000, E1   +32.851, E3 +424864.642}
SPL {X  -159.990, Y  +486.073, Z    +0.000, E1   +33.960, E3 +424877.277}
SPL {X  -159.990, Y  +477.314, Z    +0.000, E1   +35.342, E3 +424895.455}
SPL {X  -159.990, Y  +471.459, Z    +0.000, E1   +35.779, E3 +424909.995}
SPL {X  -159.990, Y  +467.485, Z    +0.000, E1   +35.768, E3 +424921.725}
SPL {X  -159.990, Y  +462.739, Z    +0.000, E1   +35.799, E3 +424935.652}
SPL {X  -159.990, Y  +457.385, Z    +0.000, E1   +35.788, E3 +424951.436}
SPL {X  -159.990, Y  +452.637, Z    +0.000, E1   +35.783, E3 +424965.428}
SPL {X  -159.990, Y  +448.227, Z    +0.000, E1   +35.776, E3 +424978.424}
SPL {X  -159.990, Y  +443.707, Z    +0.000, E1   +35.784, E3 +424991.720}
SPL {X  -159.990, Y  +439.109, Z    +0.000, E1   +35.781, E3 +425005.255}
SPL {X  -159.990, Y  +434.400, Z    +0.000, E1   +35.789, E3 +425019.110}
SPL {X  -159.990, Y  +430.115, Z    +0.000, E1   +35.777, E3 +425031.727}
SPL {X  -159.990, Y  +425.407, Z    +0.000, E1   +35.800, E3 +425045.567}
SPL {X  -159.990, Y  +420.199, Z    +0.000, E1   +35.790, E3 +425060.921}
SPL {X  -159.990, Y  +414.514, Z    +0.000, E1   +35.815, E3 +425077.620}
SPL {X  -159.990, Y  +408.600, Z    +0.000, E1   +35.802, E3 +425095.058}
SPL {X  -159.990, Y  +403.496, Z    +0.000, E1   +35.787, E3 +425110.113}
SPL {X  -159.990, Y  +398.606, Z    +0.000, E1   +35.794, E3 +425124.501}
SPL {X  -159.990, Y  +394.138, Z    +0.000, E1   +35.778, E3 +425137.684}
SPL {X  -159.990, Y  +388.813, Z    +0.000, E1   +35.819, E3 +425153.296}
SPL {X  -159.990, Y  +383.172, Z    +0.000, E1   +35.789, E3 +425169.950}
SPL {X  -159.936, Y  +378.352, Z    +0.000, E1   +35.782, E3 +425184.189}
SPL {X  -159.693, Y  +372.749, Z    +0.000, E1   +35.767, E3 +425200.921}
SPL {X  -159.203, Y  +366.647, Z    +0.000, E1   +35.680, E3 +425219.407}
SPL {X  -158.715, Y  +362.338, Z    +0.000, E1   +35.547, E3 +425232.712}
SPL {X  -158.237, Y  +358.884, Z    +0.000, E1   +35.480, E3 +425243.369}
SPL {X  -157.724, Y  +355.670, Z    +0.000, E1   +35.371, E3 +425253.403}
SPL {X  -157.185, Y  +352.671, Z    +0.000, E1   +35.292, E3 +425262.782}
SPL {X  -156.302, Y  +348.345, Z    +0.000, E1   +35.165, E3 +425276.403}
SPL {X  -155.054, Y  +343.066, Z    +0.000, E1   +34.964, E3 +425293.217}
SPL {X  -154.305, Y  +340.232, Z    +0.000, E1   +28.975, E3 +425350.777}
ENDSPLINE

SPLINE
SPL {X  -158.456, Y  +360.399, Z    +0.000, E1   +16.490, E3 +425387.597}
SPL {X  -159.553, Y  +370.677, Z    +0.000, E1   +10.576, E3 +425395.357}
SPL {X  -159.960, Y  +379.402, Z    +0.000, E1    +5.303, E3 +425399.377}
SPL {X  -159.990, Y  +387.301, Z    +0.000, E1    +0.001, E3 +425401.839}
SPL {X  -159.990, Y  +392.161, Z    +0.000, E1    -3.946, E3 +425403.250}
SPL {X  -159.990, Y  +396.375, Z    +0.000, E1    -7.538, E3 +425404.672}
SPL {X  -159.990, Y  +404.277, Z    +0.000, E1   -14.543, E3 +425408.335}
SPL {X  -159.990, Y  +423.101, Z    +0.000, E1   -27.351, E3 +425424.774}
SPL {X  -159.990, Y  +430.933, Z    +0.000, E1   -30.672, E3 +425434.745}
SPL {X  -159.990, Y  +451.842, Z    +0.000, E1   -35.050, E3 +425474.117}
SPL {X  -159.990, Y  +456.402, Z    +0.000, E1   -35.061, E3 +425487.892}
SPL {X  -159.990, Y  +460.708, Z    +0.000, E1   -35.045, E3 +425500.950}
SPL {X  -159.990, Y  +464.162, Z    +0.000, E1   -35.038, E3 +425511.407}
SPL {X  -159.990, Y  +467.857, Z    +0.000, E1   -35.053, E3 +425522.563}
SPL {X  -159.990, Y  +471.326, Z    +0.000, E1   -35.038, E3 +425533.059}
SPL {X  -159.990, Y  +474.610, Z    +0.000, E1   -35.053, E3 +425542.958}
SPL {X  -159.990, Y  +478.303, Z    +0.000, E1   -35.049, E3 +425554.130}
SPL {X  -159.990, Y  +482.537, Z    +0.000, E1   -35.066, E3 +425566.922}
SPL {X  -159.990, Y  +487.181, Z    +0.000, E1   -35.054, E3 +425581.004}
SPL {X  -159.990, Y  +492.368, Z    +0.000, E1   -35.076, E3 +425596.676}
SPL {X  -159.990, Y  +497.072, Z    +0.000, E1   -35.040, E3 +425610.973}
SPL {X  -159.990, Y  +501.645, Z    +0.000, E1   -35.067, E3 +425624.756}
SPL {X  -159.990, Y  +506.307, Z    +0.000, E1   -35.049, E3 +425638.878}
SPL {X  -159.990, Y  +511.643, Z    +0.000, E1   -35.091, E3 +425654.958}
SPL {X  -159.990, Y  +517.156, Z    +0.000, E1   -35.059, E3 +425671.676}
SPL {X  -159.990, Y  +521.637, Z    +0.000, E1   -35.056, E3 +425685.239}
SPL {X  -159.990, Y  +526.246, Z    +0.000, E1   -35.065, E3 +425699.143}
SPL {X  -159.990, Y  +530.289, Z    +0.000, E1   -35.044, E3 +425711.429}
SPL {X  -159.990, Y  +534.797, Z    +0.000, E1   -35.069, E3 +425725.029}
SPL {X  -159.990, Y  +538.710, Z    +0.000, E1   -35.033, E3 +425736.926}
SPL {X  -159.990, Y  +542.114, Z    +0.000, E1   -35.053, E3 +425747.178}
SPL {X  -159.990, Y  +545.724, Z    +0.000, E1   -35.043, E3 +425758.103}
SPL {X  -159.990, Y  +549.546, Z    +0.000, E1   -35.061, E3 +425769.627}
SPL {X  -159.990, Y  +554.793, Z    +0.000, E1   -35.100, E3 +425785.390}
SPL {X  -159.990, Y  +560.931, Z    +0.000, E1   -35.098, E3 +425803.952}
SPL {X  -159.990, Y  +566.542, Z    +0.000, E1   -35.080, E3 +425820.959}
SPL {X  -159.990, Y  +570.261, Z    +0.000, E1   -35.046, E3 +425832.256}
SPL {X  -159.990, Y  +574.780, Z    +0.000, E1   -35.101, E3 +425845.835}
SPL {X  -159.990, Y  +580.750, Z    +0.000, E1   -35.087, E3 +425863.911}
SPL {X  -159.990, Y  +585.414, Z    +0.000, E1   -35.059, E3 +425878.057}
SPL {X  -159.990, Y  +588.716, Z    +0.000, E1   -35.047, E3 +425888.060}
SPL {X  -159.990, Y  +592.923, Z    +0.000, E1   -35.084, E3 +425900.724}
SPL {X  -159.990, Y  +598.554, Z    +0.000, E1   -35.088, E3 +425917.743}
SPL {X  -159.990, Y  +603.289, Z    +0.000, E1   -35.068, E3 +425932.071}
SPL {X  -159.990, Y  +606.793, Z    +0.000, E1   -35.050, E3 +425942.713}
SPL {X  -159.990, Y  +611.113, Z    +0.000, E1   -35.087, E3 +425955.704}
SPL {X  -159.990, Y  +616.690, Z    +0.000, E1   -35.089, E3 +425972.567}
SPL {X  -159.990, Y  +621.534, Z    +0.000, E1   -35.068, E3 +425987.226}
SPL {X  -159.990, Y  +625.237, Z    +0.000, E1   -35.062, E3 +425998.428}
SPL {X  -159.990, Y  +629.217, Z    +0.000, E1   -35.065, E3 +426010.486}
SPL {X  -159.990, Y  +632.566, Z    +0.000, E1   -35.044, E3 +426020.648}
SPL {X  -159.990, Y  +636.917, Z    +0.000, E1   -35.095, E3 +426033.723}
SPL {X  -159.990, Y  +641.534, Z    +0.000, E1   -35.053, E3 +426047.750}
SPL {X  -159.990, Y  +645.423, Z    +0.000, E1   -35.070, E3 +426059.486}
SPL {X  -159.990, Y  +650.555, Z    +0.000, E1   -35.089, E3 +426074.975}
SPL {X  -159.990, Y  +656.270, Z    +0.000, E1   -35.087, E3 +426092.268}
SPL {X  -159.990, Y  +661.105, Z    +0.000, E1   -35.059, E3 +426106.932}
SPL {X  -159.990, Y  +665.311, Z    +0.000, E1   -35.064, E3 +426119.646}
SPL {X  -159.990, Y  +670.193, Z    +0.000, E1   -35.076, E3 +426134.393}
SPL {X  -159.948, Y  +675.148, Z    +0.000, E1   -35.069, E3 +426149.385}
SPL {X  -159.805, Y  +679.202, Z    +0.000, E1   -35.029, E3 +426161.818}
SPL {X  -159.584, Y  +682.885, Z    +0.000, E1   -34.997, E3 +426173.178}
SPL {X  -159.292, Y  +686.426, Z    +0.000, E1   -34.947, E3 +426184.180}
SPL {X  -158.886, Y  +690.264, Z    +0.000, E1   -34.888, E3 +426196.196}
SPL {X  -158.362, Y  +694.266, Z    +0.000, E1   -34.794, E3 +426208.870}
SPL {X  -157.614, Y  +698.973, Z    +0.000, E1   -34.690, E3 +426223.870}
SPL {X  -156.640, Y  +704.066, Z    +0.000, E1   -34.516, E3 +426240.295}
SPL {X  -155.835, Y  +707.723, Z    +0.000, E1   -34.344, E3 +426252.238}
SPL {X  -155.153, Y  +710.542, Z    +0.000, E1   -34.234, E3 +426261.457}
SPL {X  -153.767, Y  +715.686, Z    +0.000, E1   -30.747, E3 +426306.675}
ENDSPLINE

SPLINE
SPL {X  -155.537, Y  +708.983, Z    +0.000, E1   -25.008, E3 +426337.480}
SPL {X  -158.838, Y  +690.666, Z    +0.000, E1   -14.584, E3 +426362.193}
SPL {X  -159.750, Y  +680.262, Z    +0.000, E1    -8.563, E3 +426368.333}
SPL {X  -159.973, Y  +673.798, Z    +0.000, E1    -4.600, E3 +426370.797}
SPL {X  -159.990, Y  +667.448, Z    +0.000, E1    -0.356, E3 +426372.577}
SPL {X  -159.990, Y  +662.686, Z    +0.000, E1    +3.472, E3 +426373.812}
SPL {X  -159.990, Y  +657.071, Z    +0.000, E1    +8.297, E3 +426375.690}
SPL {X  -159.990, Y  +646.193, Z    +0.000, E1   +17.980, E3 +426381.417}
SPL {X  -159.990, Y  +621.124, Z    +0.000, E1   +32.598, E3 +426404.903}
SPL {X  -159.990, Y  +597.855, Z    +0.000, E1   +36.862, E3 +426447.823}
SPL {X  -159.990, Y  +592.884, Z    +0.000, E1   +36.865, E3 +426461.894}
SPL {X  -159.990, Y  +587.104, Z    +0.000, E1   +36.878, E3 +426478.250}
SPL {X  -159.990, Y  +581.795, Z    +0.000, E1   +36.847, E3 +426493.349}
SPL {X  -159.990, Y  +577.286, Z    +0.000, E1   +36.853, E3 +426506.106}
SPL {X  -159.990, Y  +572.409, Z    +0.000, E1   +36.854, E3 +426519.918}
SPL {X  -159.990, Y  +567.110, Z    +0.000, E1   +36.868, E3 +426534.880}
SPL {X  -159.990, Y  +562.387, Z    +0.000, E1   +36.853, E3 +426548.241}
SPL {X  -159.990, Y  +557.944, Z    +0.000, E1   +36.859, E3 +426560.835}
SPL {X  -159.990, Y  +553.661, Z    +0.000, E1   +36.844, E3 +426572.998}
SPL {X  -159.990, Y  +549.195, Z    +0.000, E1   +36.856, E3 +426585.633}
SPL {X  -159.990, Y  +544.733, Z    +0.000, E1   +36.845, E3 +426598.279}
SPL {X  -159.990, Y  +539.889, Z    +0.000, E1   +36.872, E3 +426611.964}
SPL {X  -159.990, Y  +534.469, Z    +0.000, E1   +36.855, E3 +426627.361}
SPL {X  -159.990, Y  +530.428, Z    +0.000, E1   +36.821, E3 +426638.895}
SPL {X  -159.990, Y  +527.151, Z    +0.000, E1   +36.828, E3 +426648.158}
SPL {X  -159.990, Y  +522.641, Z    +0.000, E1   +36.854, E3 +426660.890}
SPL {X  -159.990, Y  +517.225, Z    +0.000, E1   +36.859, E3 +426676.225}
SPL {X  -159.990, Y  +512.789, Z    +0.000, E1   +36.824, E3 +426688.852}
SPL {X  -159.990, Y  +508.591, Z    +0.000, E1   +36.846, E3 +426700.715}
SPL {X  -159.990, Y  +503.454, Z    +0.000, E1   +36.847, E3 +426715.270}
SPL {X  -159.990, Y  +498.507, Z    +0.000, E1   +36.487, E3 +426731.719}
ENDSPLINE

SPLINE
SPL {X  -159.990, Y  +506.994, Z    +0.000, E1   +30.162, E3 +426744.228}
ENDSPLINE

SPLINE
SPL {X  -159.990, Y  +502.084, Z    +0.000, E1   +31.057, E3 +426755.880}
SPL {X  -159.990, Y  +496.272, Z    +0.000, E1   +32.117, E3 +426768.871}
SPL {X  -159.990, Y  +492.180, Z    +0.000, E1   +32.851, E3 +426777.685}
SPL {X  -159.990, Y  +486.073, Z    +0.000, E1   +33.960, E3 +426790.321}
SPL {X  -159.990, Y  +477.314, Z    +0.000, E1   +35.342, E3 +426808.499}
SPL {X  -159.990, Y  +471.459, Z    +0.000, E1   +35.779, E3 +426823.038}
SPL {X  -159.990, Y  +467.485, Z    +0.000, E1   +35.768, E3 +426834.768}
SPL {X  -159.990, Y  +462.739, Z    +0.000, E1   +35.799, E3 +426848.696}
SPL {X  -159.990, Y  +457.385, Z    +0.000, E1   +35.788, E3 +426864.479}
SPL {X  -159.990, Y  +452.637, Z    +0.000, E1   +35.783, E3 +426878.471}
SPL {X  -159.990, Y  +448.227, Z    +0.000, E1   +35.776, E3 +426891.468}
SPL {X  -159.990, Y  +443.707, Z    +0.000, E1   +35.784, E3 +426904.763}
SPL {X  -159.990, Y  +439.109, Z    +0.000, E1   +35.781, E3 +426918.299}
SPL {X  -159.990, Y  +435.535, Z    +0.000, E1   +35.764, E3 +426928.849}
SPL {X  -159.990, Y  +431.100, Z    +0.000, E1   +35.807, E3 +426941.835}
SPL {X  -159.990, Y  +426.641, Z    +0.000, E1   +35.769, E3 +426955.021}
SPL {X  -159.990, Y  +422.627, Z    +0.000, E1   +35.788, E3 +426966.819}
SPL {X  -159.990, Y  +419.027, Z    +0.000, E1   +35.762, E3 +426977.459}
SPL {X  -159.990, Y  +414.514, Z    +0.000, E1   +35.815, E3 +426990.663}
SPL {X  -159.990, Y  +409.702, Z    +0.000, E1   +35.772, E3 +427004.904}
SPL {X  -159.990, Y  +404.413, Z    +0.000, E1   +35.821, E3 +427020.406}
SPL {X  -159.990, Y  +398.606, Z    +0.000, E1   +35.794, E3 +427037.544}
SPL {X  -159.990, Y  +394.138, Z    +0.000, E1   +35.778, E3 +427050.727}
SPL {X  -159.990, Y  +388.813, Z    +0.000, E1   +35.819, E3 +427066.339}
SPL {X  -159.990, Y  +383.172, Z    +0.000, E1   +35.789, E3 +427082.993}
SPL {X  -159.936, Y  +378.352, Z    +0.000, E1   +35.782, E3 +427097.232}
SPL {X  -159.790, Y  +374.497, Z    +0.000, E1   +35.735, E3 +427108.777}
SPL {X  -159.547, Y  +370.604, Z    +0.000, E1   +35.724, E3 +427120.462}
SPL {X  -159.134, Y  +365.969, Z    +0.000, E1   +35.644, E3 +427134.547}
SPL {X  -158.606, Y  +361.498, Z    +0.000, E1   +35.550, E3 +427148.312}
SPL {X  -157.918, Y  +356.833, Z    +0.000, E1   +35.439, E3 +427162.764}
SPL {X  -157.185, Y  +352.671, Z    +0.000, E1   +35.292, E3 +427175.825}
SPL {X  -156.302, Y  +348.345, Z    +0.000, E1   +35.165, E3 +427189.446}
SPL {X  -155.054, Y  +343.066, Z    +0.000, E1   +34.964, E3 +427206.261}
SPL {X  -154.305, Y  +340.232, Z    +0.000, E1   +28.975, E3 +427263.821}
ENDSPLINE

SPLINE
SPL {X  -158.456, Y  +360.399, Z    +0.000, E1   +16.490, E3 +427300.640}
SPL {X  -159.553, Y  +370.677, Z    +0.000, E1   +10.576, E3 +427308.401}
SPL {X  -159.960, Y  +379.402, Z    +0.000, E1    +5.303, E3 +427312.421}
SPL {X  -159.990, Y  +387.301, Z    +0.000, E1    +0.001, E3 +427314.882}
SPL {X  -159.990, Y  +392.161, Z    +0.000, E1    -3.946, E3 +427316.294}
SPL {X  -159.990, Y  +396.375, Z    +0.000, E1    -7.538, E3 +427317.716}
SPL {X  -159.990, Y  +404.277, Z    +0.000, E1   -14.543, E3 +427321.379}
SPL {X  -159.990, Y  +423.101, Z    +0.000, E1   -27.351, E3 +427337.818}
SPL {X  -159.990, Y  +430.933, Z    +0.000, E1   -30.672, E3 +427347.788}
SPL {X  -159.990, Y  +452.779, Z    +0.000, E1   -35.077, E3 +427389.952}
SPL {X  -159.990, Y  +457.209, Z    +0.000, E1   -35.039, E3 +427403.411}
SPL {X  -159.990, Y  +460.708, Z    +0.000, E1   -35.045, E3 +427413.994}
SPL {X  -159.990, Y  +464.162, Z    +0.000, E1   -35.038, E3 +427424.450}
SPL {X  -159.990, Y  +467.857, Z    +0.000, E1   -35.053, E3 +427435.607}
SPL {X  -159.990, Y  +471.326, Z    +0.000, E1   -35.038, E3 +427446.102}
SPL {X  -159.990, Y  +474.610, Z    +0.000, E1   -35.053, E3 +427456.002}
SPL {X  -159.990, Y  +479.424, Z    +0.000, E1   -35.081, E3 +427470.514}
SPL {X  -159.990, Y  +483.513, Z    +0.000, E1   -35.038, E3 +427482.968}
SPL {X  -159.990, Y  +487.181, Z    +0.000, E1   -35.054, E3 +427494.048}
SPL {X  -159.990, Y  +490.807, Z    +0.000, E1   -35.036, E3 +427505.049}
SPL {X  -159.990, Y  +493.669, Z    +0.000, E1   -35.034, E3 +427513.729}
SPL {X  -159.990, Y  +497.072, Z    +0.000, E1   -35.040, E3 +427524.016}
SPL {X  -159.990, Y  +500.395, Z    +0.000, E1   -35.033, E3 +427534.079}
SPL {X  -159.990, Y  +505.138, Z    +0.000, E1   -35.092, E3 +427548.315}
SPL {X  -159.990, Y  +510.443, Z    +0.000, E1   -35.051, E3 +427564.434}
SPL {X  -159.990, Y  +514.632, Z    +0.000, E1   -35.050, E3 +427577.104}
SPL {X  -159.990, Y  +518.055, Z    +0.000, E1   -35.037, E3 +427587.473}
SPL {X  -159.990, Y  +521.637, Z    +0.000, E1   -35.056, E3 +427598.283}
SPL {X  -159.990, Y  +526.246, Z    +0.000, E1   -35.065, E3 +427612.186}
SPL {X  -159.990, Y  +531.319, Z    +0.000, E1   -35.072, E3 +427627.542}
SPL {X  -159.990, Y  +537.053, Z    +0.000, E1   -35.083, E3 +427644.875}
SPL {X  -159.990, Y  +542.114, Z    +0.000, E1   -35.053, E3 +427660.222}
SPL {X  -159.990, Y  +546.612, Z    +0.000, E1   -35.065, E3 +427673.793}
SPL {X  -159.990, Y  +551.596, Z    +0.000, E1   -35.079, E3 +427688.828}
SPL {X  -159.990, Y  +557.043, Z    +0.000, E1   -35.087, E3 +427705.250}
SPL {X  -159.990, Y  +561.808, Z    +0.000, E1   -35.066, E3 +427719.703}
SPL {X  -159.990, Y  +566.542, Z    +0.000, E1   -35.080, E3 +427734.003}
SPL {X  -159.990, Y  +571.374, Z    +0.000, E1   -35.070, E3 +427748.627}
SPL {X  -159.990, Y  +575.771, Z    +0.000, E1   -35.064, E3 +427761.932}
SPL {X  -159.990, Y  +580.750, Z    +0.000, E1   -35.087, E3 +427776.954}
SPL {X  -159.990, Y  +585.414, Z    +0.000, E1   -35.059, E3 +427791.101}
SPL {X  -159.990, Y  +590.166, Z    +0.000, E1   -35.084, E3 +427805.429}
SPL {X  -159.990, Y  +595.313, Z    +0.000, E1   -35.073, E3 +427821.008}
SPL {X  -159.990, Y  +600.543, Z    +0.000, E1   -35.091, E3 +427836.790}
SPL {X  -159.990, Y  +605.846, Z    +0.000, E1   -35.077, E3 +427852.841}
SPL {X  -159.990, Y  +611.113, Z    +0.000, E1   -35.087, E3 +427868.747}
SPL {X  -159.990, Y  +616.690, Z    +0.000, E1   -35.089, E3 +427885.611}
SPL {X  -159.990, Y  +621.534, Z    +0.000, E1   -35.068, E3 +427900.270}
SPL {X  -159.990, Y  +626.426, Z    +0.000, E1   -35.093, E3 +427915.029}
SPL {X  -159.990, Y  +631.553, Z    +0.000, E1   -35.068, E3 +427930.587}
SPL {X  -159.990, Y  +635.965, Z    +0.000, E1   -35.065, E3 +427943.935}
SPL {X  -159.990, Y  +640.633, Z    +0.000, E1   -35.080, E3 +427958.024}
SPL {X  -159.990, Y  +645.423, Z    +0.000, E1   -35.070, E3 +427972.529}
SPL {X  -159.990, Y  +650.555, Z    +0.000, E1   -35.089, E3 +427988.018}
SPL {X  -159.990, Y  +656.270, Z    +0.000, E1   -35.087, E3 +428005.311}
SPL {X  -159.990, Y  +661.105, Z    +0.000, E1   -35.059, E3 +428019.975}
SPL {X  -159.990, Y  +665.311, Z    +0.000, E1   -35.064, E3 +428032.690}
SPL {X  -159.990, Y  +670.193, Z    +0.000, E1   -35.076, E3 +428047.437}
SPL {X  -159.948, Y  +675.148, Z    +0.000, E1   -35.069, E3 +428062.429}
SPL {X  -159.752, Y  +680.228, Z    +0.000, E1   -35.050, E3 +428077.977}
SPL {X  -159.371, Y  +685.563, Z    +0.000, E1   -34.989, E3 +428094.488}
SPL {X  -158.886, Y  +690.264, Z    +0.000, E1   -34.888, E3 +428109.240}
SPL {X  -158.362, Y  +694.266, Z    +0.000, E1   -34.794, E3 +428121.913}
SPL {X  -157.614, Y  +698.973, Z    +0.000, E1   -34.690, E3 +428136.914}
SPL {X  -156.640, Y  +704.066, Z    +0.000, E1   -34.516, E3 +428153.339}
SPL {X  -155.835, Y  +707.723, Z    +0.000, E1   -34.344, E3 +428165.281}
SPL {X  -155.153, Y  +710.542, Z    +0.000, E1   -34.234, E3 +428174.501}
SPL {X  -153.767, Y  +715.686, Z    +0.000, E1   -30.747, E3 +428219.719}
ENDSPLINE

SPLINE
SPL {X  -155.537, Y  +708.983, Z    +0.000, E1   -25.008, E3 +428250.523}
SPL {X  -158.838, Y  +690.666, Z    +0.000, E1   -14.584, E3 +428275.236}
SPL {X  -159.750, Y  +680.262, Z    +0.000, E1    -8.563, E3 +428281.377}
SPL {X  -159.973, Y  +673.798, Z    +0.000, E1    -4.600, E3 +428283.840}
SPL {X  -159.990, Y  +668.863, Z    +0.000, E1    -1.298, E3 +428285.280}
SPL {X  -159.990, Y  +663.839, Z    +0.000, E1    +2.454, E3 +428286.541}
SPL {X  -159.990, Y  +658.349, Z    +0.000, E1    +7.223, E3 +428288.223}
SPL {X  -159.990, Y  +650.390, Z    +0.000, E1   +14.372, E3 +428291.969}
SPL {X  -159.990, Y  +643.417, Z    +0.000, E1   +20.300, E3 +428296.233}
SPL {X  -159.990, Y  +621.124, Z    +0.000, E1   +32.598, E3 +428317.947}
SPL {X  -159.990, Y  +597.855, Z    +0.000, E1   +36.862, E3 +428360.866}
SPL {X  -159.990, Y  +592.884, Z    +0.000, E1   +36.865, E3 +428374.937}
SPL {X  -159.990, Y  +587.104, Z    +0.000, E1   +36.878, E3 +428391.294}
SPL {X  -159.990, Y  +581.795, Z    +0.000, E1   +36.847, E3 +428406.393}
SPL {X  -159.990, Y  +577.286, Z    +0.000, E1   +36.853, E3 +428419.149}
SPL {X  -159.990, Y  +572.409, Z    +0.000, E1   +36.854, E3 +428432.962}
SPL {X  -159.990, Y  +567.110, Z    +0.000, E1   +36.868, E3 +428447.923}
SPL {X  -159.990, Y  +562.387, Z    +0.000, E1   +36.853, E3 +428461.284}
SPL {X  -159.990, Y  +557.944, Z    +0.000, E1   +36.859, E3 +428473.878}
SPL {X  -159.990, Y  +552.571, Z    +0.000, E1   +36.873, E3 +428489.082}
SPL {X  -159.990, Y  +546.127, Z    +0.000, E1   +36.890, E3 +428507.309}
SPL {X  -159.990, Y  +539.889, Z    +0.000, E1   +36.872, E3 +428525.007}
SPL {X  -159.990, Y  +534.469, Z    +0.000, E1   +36.855, E3 +428540.405}
SPL {X  -159.990, Y  +528.569, Z    +0.000, E1   +36.871, E3 +428557.123}
SPL {X  -159.990, Y  +522.641, Z    +0.000, E1   +36.854, E3 +428573.934}
SPL {X  -159.990, Y  +517.225, Z    +0.000, E1   +36.859, E3 +428589.268}
SPL {X  -159.990, Y  +511.408, Z    +0.000, E1   +36.858, E3 +428605.756}
SPL {X  -159.990, Y  +505.756, Z    +0.000, E1   +36.857, E3 +428621.766}
SPL {X  -159.990, Y  +499.829, Z    +0.000, E1   +36.864, E3 +428638.571}
SPL {X  -159.990, Y  +498.054, Z    +0.000, E1   +35.692, E3 +428650.610}
ENDSPLINE

SPLINE
SPL {X  -159.990, Y  +506.994, Z    +0.000, E1   +30.162, E3 +428657.272}
ENDSPLINE

SPLINE
SPL {X  -159.990, Y  +502.084, Z    +0.000, E1   +31.057, E3 +428668.923}
SPL {X  -159.990, Y  +494.586, Z    +0.000, E1   +32.444, E3 +428685.526}
SPL {X  -159.990, Y  +486.073, Z    +0.000, E1   +33.960, E3 +428703.364}
SPL {X  -159.990, Y  +477.312, Z    +0.000, E1   +35.343, E3 +428721.542}
ENDSPLINE

SPLINE
SPL {X  -159.990, Y  +491.651, Z    +0.000, E1   +25.403, E3 +428736.613}
ENDSPLINE

SPLINE
SPL {X  -159.990, Y  +488.807, Z    +0.000, E1   +25.397, E3 +428749.338}
SPL {X  -159.990, Y  +486.070, Z    +0.000, E1   +25.399, E3 +428761.569}
SPL {X  -159.990, Y  +482.821, Z    +0.000, E1   +25.411, E3 +428776.070}
SPL {X  -159.990, Y  +480.183, Z    +0.000, E1   +25.384, E3 +428787.911}
SPL {X  -159.990, Y  +477.508, Z    +0.000, E1   +25.410, E3 +428799.819}
SPL {X  -159.990, Y  +473.634, Z    +0.000, E1   +25.426, E3 +428817.108}
SPL {X  -159.990, Y  +470.047, Z    +0.000, E1   +25.402, E3 +428833.189}
SPL {X  -159.990, Y  +466.213, Z    +0.000, E1   +25.433, E3 +428850.269}
SPL {X  -159.990, Y  +462.520, Z    +0.000, E1   +25.400, E3 +428866.838}
SPL {X  -159.990, Y  +460.081, Z    +0.000, E1   +25.390, E3 +428877.739}
SPL {X  -159.990, Y  +457.497, Z    +0.000, E1   +25.403, E3 +428889.264}
SPL {X  -159.990, Y  +455.126, Z    +0.000, E1   +25.389, E3 +428899.872}
SPL {X  -159.990, Y  +452.123, Z    +0.000, E1   +25.426, E3 +428913.230}
SPL {X  -159.990, Y  +448.503, Z    +0.000, E1   +25.410, E3 +428929.431}
SPL {X  -159.990, Y  +445.882, Z    +0.000, E1   +25.385, E3 +428941.234}
SPL {X  -159.990, Y  +443.345, Z    +0.000, E1   +25.390, E3 +428952.616}
SPL {X  -159.990, Y  +440.220, Z    +0.000, E1   +25.392, E3 +428966.603}
SPL {X  -159.990, Y  +436.316, Z    +0.000, E1   +25.420, E3 +428984.007}
SPL {X  -159.990, Y  +432.613, Z    +0.000, E1   +25.390, E3 +429000.632}
SPL {X  -159.990, Y  +429.827, Z    +0.000, E1   +25.380, E3 +429013.110}
SPL {X  -159.990, Y  +426.865, Z    +0.000, E1   +25.398, E3 +429026.314}
SPL {X  -159.990, Y  +423.417, Z    +0.000, E1   +25.400, E3 +429041.730}
SPL {X  -159.990, Y  +420.283, Z    +0.000, E1   +25.386, E3 +429055.775}
SPL {X  -159.990, Y  +417.514, Z    +0.000, E1   +25.386, E3 +429068.159}
SPL {X  -159.990, Y  +414.805, Z    +0.000, E1   +25.385, E3 +429080.280}
SPL {X  -159.990, Y  +411.959, Z    +0.000, E1   +25.386, E3 +429093.006}
SPL {X  -159.990, Y  +408.981, Z    +0.000, E1   +25.392, E3 +429106.310}
SPL {X  -159.990, Y  +405.773, Z    +0.000, E1   +25.398, E3 +429120.620}
SPL {X  -159.990, Y  +402.805, Z    +0.000, E1   +25.389, E3 +429133.906}
SPL {X  -159.990, Y  +400.083, Z    +0.000, E1   +25.388, E3 +429146.083}
SPL {X  -159.990, Y  +396.740, Z    +0.000, E1   +25.410, E3 +429161.007}
SPL {X  -159.990, Y  +392.622, Z    +0.000, E1   +25.413, E3 +429179.435}
SPL {X  -159.990, Y  +388.328, Z    +0.000, E1   +25.413, E3 +429198.663}
SPL {X  -159.990, Y  +384.900, Z    +0.000, E1   +25.383, E3 +429214.025}
SPL {X  -159.990, Y  +382.110, Z    +0.000, E1   +25.393, E3 +429226.472}
SPL {X  -159.961, Y  +379.439, Z    +0.000, E1   +25.380, E3 +429238.451}
SPL {X  -159.894, Y  +376.959, Z    +0.000, E1   +25.370, E3 +429249.629}
SPL {X  -159.784, Y  +374.382, Z    +0.000, E1   +25.356, E3 +429261.269}
SPL {X  -159.621, Y  +371.640, Z    +0.000, E1   +25.335, E3 +429273.709}
SPL {X  -159.406, Y  +368.844, Z    +0.000, E1   +25.307, E3 +429286.422}
SPL {X  -159.144, Y  +366.072, Z    +0.000, E1   +25.281, E3 +429299.030}
SPL {X  -158.822, Y  +363.200, Z    +0.000, E1   +25.236, E3 +429312.202}
SPL {X  -158.491, Y  +360.654, Z    +0.000, E1   +25.188, E3 +429323.942}
SPL {X  -158.127, Y  +358.155, Z    +0.000, E1   +25.126, E3 +429335.562}
SPL {X  -158.095, Y  +357.947, Z    +0.000, E1   +21.741, E3 +429367.134}
ENDSPLINE

SPLINE
SPL {X  -158.454, Y  +360.384, Z    +0.000, E1   +19.366, E3 +429379.285}
SPL {X  -159.737, Y  +373.507, Z    +0.000, E1   +10.311, E3 +429401.321}
SPL {X  -159.990, Y  +382.574, Z    +0.000, E1    +4.463, E3 +429408.008}
SPL {X  -159.990, Y  +387.496, Z    +0.000, E1    +1.004, E3 +429410.754}
SPL {X  -159.990, Y  +395.121, Z    +0.000, E1    -4.514, E3 +429415.066}
SPL {X  -159.990, Y  +407.941, Z    +0.000, E1   -14.126, E3 +429427.140}
SPL {X  -159.990, Y  +418.671, Z    +0.000, E1   -19.855, E3 +429446.556}
SPL {X  -159.990, Y  +429.878, Z    +0.000, E1   -23.330, E3 +429476.611}
SPL {X  -159.990, Y  +432.766, Z    +0.000, E1   -23.321, E3 +429490.834}
SPL {X  -159.990, Y  +434.794, Z    +0.000, E1   -23.304, E3 +429500.865}
SPL {X  -159.990, Y  +437.007, Z    +0.000, E1   -23.323, E3 +429511.718}
SPL {X  -159.990, Y  +439.778, Z    +0.000, E1   -23.323, E3 +429525.350}
SPL {X  -159.990, Y  +442.010, Z    +0.000, E1   -23.308, E3 +429536.371}
SPL {X  -159.990, Y  +443.729, Z    +0.000, E1   -23.310, E3 +429544.827}
SPL {X  -159.990, Y  +446.037, Z    +0.000, E1   -23.324, E3 +429556.164}
SPL {X  -159.990, Y  +449.434, Z    +0.000, E1   -23.356, E3 +429572.786}
SPL {X  -159.990, Y  +453.256, Z    +0.000, E1   -23.349, E3 +429591.621}
SPL {X  -159.990, Y  +455.953, Z    +0.000, E1   -23.320, E3 +429604.935}
SPL {X  -159.990, Y  +458.265, Z    +0.000, E1   -23.328, E3 +429616.289}
SPL {X  -159.990, Y  +460.492, Z    +0.000, E1   -23.317, E3 +429627.288}
SPL {X  -159.990, Y  +462.929, Z    +0.000, E1   -23.331, E3 +429639.244}
SPL {X  -159.990, Y  +466.197, Z    +0.000, E1   -23.351, E3 +429655.281}
SPL {X  -159.990, Y  +468.951, Z    +0.000, E1   -23.319, E3 +429668.899}
SPL {X  -159.990, Y  +470.991, Z    +0.000, E1   -23.322, E3 +429678.928}
SPL {X  -159.990, Y  +474.027, Z    +0.000, E1   -23.352, E3 +429693.832}
SPL {X  -159.990, Y  +476.830, Z    +0.000, E1   -23.323, E3 +429707.700}
SPL {X  -159.990, Y  +479.553, Z    +0.000, E1   -23.328, E3 +429721.102}
SPL {X  -159.990, Y  +482.950, Z    +0.000, E1   -23.350, E3 +429737.774}
SPL {X  -159.990, Y  +486.109, Z    +0.000, E1   -23.322, E3 +429753.390}
SPL {X  -159.990, Y  +488.481, Z    +0.000, E1   -23.319, E3 +429765.070}
SPL {X  -159.990, Y  +491.454, Z    +0.000, E1   -23.343, E3 +429779.650}
SPL {X  -159.990, Y  +494.937, Z    +0.000, E1   -23.343, E3 +429796.794}
SPL {X  -159.990, Y  +497.668, Z    +0.000, E1   -23.317, E3 +429810.287}
SPL {X  -159.990, Y  +499.995, Z    +0.000, E1   -23.324, E3 +429821.725}
SPL {X  -159.990, Y  +502.456, Z    +0.000, E1   -23.324, E3 +429833.840}
SPL {X  -159.990, Y  +505.646, Z    +0.000, E1   -23.350, E3 +429849.495}
SPL {X  -159.990, Y  +508.862, Z    +0.000, E1   -23.328, E3 +429865.359}
SPL {X  -159.990, Y  +510.971, Z    +0.000, E1   -23.308, E3 +429875.787}
SPL {X  -159.990, Y  +512.484, Z    +0.000, E1   -23.309, E3 +429883.236}
SPL {X  -159.990, Y  +514.757, Z    +0.000, E1   -23.329, E3 +429894.389}
SPL {X  -159.990, Y  +517.536, Z    +0.000, E1   -23.326, E3 +429908.055}
SPL {X  -159.990, Y  +519.961, Z    +0.000, E1   -23.334, E3 +429919.908}
SPL {X  -159.990, Y  +521.849, Z    +0.000, E1   -23.320, E3 +429929.230}
SPL {X  -159.990, Y  +523.968, Z    +0.000, E1   -23.332, E3 +429939.666}
SPL {X  -159.990, Y  +526.466, Z    +0.000, E1   -23.320, E3 +429952.009}
SPL {X  -159.990, Y  +528.815, Z    +0.000, E1   -23.322, E3 +429963.569}
SPL {X  -159.990, Y  +531.246, Z    +0.000, E1   -23.325, E3 +429975.507}
SPL {X  -159.990, Y  +534.143, Z    +0.000, E1   -23.341, E3 +429989.742}
SPL {X  -159.990, Y  +537.024, Z    +0.000, E1   -23.321, E3 +430003.986}
SPL {X  -159.990, Y  +539.129, Z    +0.000, E1   -23.310, E3 +430014.369}
SPL {X  -159.990, Y  +541.882, Z    +0.000, E1   -23.346, E3 +430027.850}
SPL {X  -159.990, Y  +544.941, Z    +0.000, E1   -23.325, E3 +430042.932}
SPL {X  -159.990, Y  +547.390, Z    +0.000, E1   -23.325, E3 +430054.986}
SPL {X  -159.990, Y  +550.708, Z    +0.000, E1   -23.357, E3 +430071.253}
SPL {X  -159.990, Y  +553.642, Z    +0.000, E1   -23.319, E3 +430085.760}
SPL {X  -159.990, Y  +555.637, Z    +0.000, E1   -23.323, E3 +430095.574}
SPL {X  -159.990, Y  +558.758, Z    +0.000, E1   -23.351, E3 +430110.884}
SPL {X  -159.990, Y  +561.830, Z    +0.000, E1   -23.325, E3 +430126.057}
SPL {X  -159.990, Y  +564.273, Z    +0.000, E1   -23.325, E3 +430138.081}
SPL {X  -159.990, Y  +567.351, Z    +0.000, E1   -23.348, E3 +430153.177}
SPL {X  -159.990, Y  +570.560, Z    +0.000, E1   -23.333, E3 +430169.007}
SPL {X  -159.990, Y  +572.975, Z    +0.000, E1   -23.316, E3 +430180.926}
SPL {X  -159.990, Y  +575.097, Z    +0.000, E1   -23.325, E3 +430191.353}
SPL {X  -159.990, Y  +577.540, Z    +0.000, E1   -23.325, E3 +430203.382}
SPL {X  -159.990, Y  +580.312, Z    +0.000, E1   -23.340, E3 +430216.963}
SPL {X  -159.990, Y  +583.018, Z    +0.000, E1   -23.331, E3 +430230.268}
SPL {X  -159.990, Y  +585.165, Z    +0.000, E1   -23.322, E3 +430240.884}
SPL {X  -159.990, Y  +587.388, Z    +0.000, E1   -23.328, E3 +430251.796}
SPL {X  -159.990, Y  +589.763, Z    +0.000, E1   -23.328, E3 +430263.483}
SPL {X  -159.990, Y  +592.397, Z    +0.000, E1   -23.344, E3 +430276.364}
SPL {X  -159.990, Y  +594.928, Z    +0.000, E1   -23.334, E3 +430288.826}
SPL {X  -159.990, Y  +597.981, Z    +0.000, E1   -23.373, E3 +430303.741}
SPL {X  -159.990, Y  +600.935, Z    +0.000, E1   -23.343, E3 +430318.273}
SPL {X  -159.990, Y  +603.047, Z    +0.000, E1   -23.344, E3 +430328.659}
SPL {X  -159.990, Y  +605.187, Z    +0.000, E1   -23.344, E3 +430339.181}
SPL {X  -159.990, Y  +607.319, Z    +0.000, E1   -23.353, E3 +430349.643}
SPL {X  -159.990, Y  +610.569, Z    +0.000, E1   -23.372, E3 +430365.608}
SPL {X  -159.990, Y  +613.591, Z    +0.000, E1   -23.342, E3 +430380.537}
SPL {X  -159.990, Y  +615.604, Z    +0.000, E1   -23.330, E3 +430390.475}
SPL {X  -159.990, Y  +618.445, Z    +0.000, E1   -23.368, E3 +430404.388}
SPL {X  -159.990, Y  +621.517, Z    +0.000, E1   -23.337, E3 +430419.552}
SPL {X  -159.990, Y  +623.764, Z    +0.000, E1   -23.335, E3 +430430.603}
SPL {X  -159.990, Y  +625.941, Z    +0.000, E1   -23.337, E3 +430441.294}
SPL {X  -159.990, Y  +628.611, Z    +0.000, E1   -23.357, E3 +430454.373}
SPL {X  -159.990, Y  +631.169, Z    +0.000, E1   -23.338, E3 +430466.977}
SPL {X  -159.990, Y  +633.318, Z    +0.000, E1   -23.339, E3 +430477.566}
SPL {X  -159.990, Y  +635.650, Z    +0.000, E1   -23.339, E3 +430489.037}
SPL {X  -159.990, Y  +637.839, Z    +0.000, E1   -23.335, E3 +430499.847}
SPL {X  -159.990, Y  +640.072, Z    +0.000, E1   -23.325, E3 +430510.879}
SPL {X  -159.990, Y  +642.230, Z    +0.000, E1   -23.323, E3 +430521.561}
SPL {X  -159.990, Y  +645.287, Z    +0.000, E1   -23.340, E3 +430536.587}
SPL {X  -159.990, Y  +648.792, Z    +0.000, E1   -23.346, E3 +430553.846}
SPL {X  -159.990, Y  +652.623, Z    +0.000, E1   -23.348, E3 +430572.681}
SPL {X  -159.990, Y  +656.380, Z    +0.000, E1   -23.347, E3 +430591.175}
SPL {X  -159.990, Y  +659.180, Z    +0.000, E1   -23.314, E3 +430605.023}
SPL {X  -159.990, Y  +661.392, Z    +0.000, E1   -23.318, E3 +430615.917}
SPL {X  -159.990, Y  +663.662, Z    +0.000, E1   -23.322, E3 +430627.041}
SPL {X  -159.990, Y  +665.964, Z    +0.000, E1   -23.328, E3 +430638.332}
SPL {X  -159.990, Y  +668.989, Z    +0.000, E1   -23.359, E3 +430653.167}
SPL {X  -159.990, Y  +671.893, Z    +0.000, E1   -23.319, E3 +430667.548}
SPL {X  -159.974, Y  +673.789, Z    +0.000, E1   -23.323, E3 +430676.863}
SPL {X  -159.924, Y  +676.110, Z    +0.000, E1   -23.320, E3 +430688.348}
SPL {X  -159.845, Y  +678.302, Z    +0.000, E1   -23.298, E3 +430699.250}
SPL {X  -159.760, Y  +680.081, Z    +0.000, E1   -23.288, E3 +430708.093}
SPL {X  -159.626, Y  +682.287, Z    +0.000, E1   -23.280, E3 +430719.065}
SPL {X  -159.462, Y  +684.486, Z    +0.000, E1   -23.258, E3 +430730.065}
SPL {X  -159.246, Y  +686.911, Z    +0.000, E1   -23.230, E3 +430742.226}
SPL {X  -159.019, Y  +689.098, Z    +0.000, E1   -23.200, E3 +430753.228}
SPL {X  -158.660, Y  +692.086, Z    +0.000, E1   -23.176, E3 +430768.272}
ENDSPLINE

